LIN {X 0,Y 419.846,Z 525.532,A -85,B 0,C 180,E1 -10292.919,E2 -10292.919} C_VEL
LIN {X 0,Y 422.177,Z 533.001,A -85,B 0,C 180,E1 -10293.178,E2 -10293.178} C_VEL
LIN {X 0,Y 424.264,Z 542.34,A -85,B 0,C 180,E1 -10293.457,E2 -10293.457} C_VEL
LIN {X 0,Y 423.052,Z 632.06,A -85,B 0,C 180,E1 -10295.077,E2 -10295.077} C_VEL
LIN {X 0,Y 422.664,Z 645.822,A -85,B 0,C 180,E1 -10295.536,E2 -10295.536} C_VEL
LIN {X 0,Y 422.218,Z 658.144,A -85,B 0,C 180,E1 -10296.147,E2 -10296.147} C_VEL
LIN {X 0,Y 421.56,Z 670.212,A -85,B 0,C 180,E1 -10296.956,E2 -10296.956} C_VEL
LIN {X 0,Y 420.936,Z 680.638,A -85,B 0,C 180,E1 -10297.848,E2 -10297.848} C_VEL
LIN {X 0,Y 420.144,Z 691.488,A -85,B 0,C 180,E1 -10299.003,E2 -10299.003} C_VEL
LIN {X 0,Y 419.475,Z 700.404,A -85,B 0,C 180,E1 -10300.187,E2 -10300.187} C_VEL
LIN {X 0,Y 418.766,Z 709.277,A -85,B 0,C 180,E1 -10301.642,E2 -10301.642} C_VEL
LIN {X 0,Y 418.301,Z 715.982,A -85,B 0,C 180,E1 -10303.007,E2 -10303.007} C_VEL
LIN {X 0,Y 417.87,Z 721.394,A -85,B 0,C 180,E1 -10304.368,E2 -10304.368} C_VEL
LIN {X 0,Y 417.597,Z 725.629,A -85,B 0,C 180,E1 -10305.7,E2 -10305.7} C_VEL
LIN {X 0,Y 417.406,Z 728.908,A -85,B 0,C 180,E1 -10307.017,E2 -10307.017} C_VEL
LIN {X 0,Y 417.134,Z 732.231,A -85,B 0,C 180,E1 -10308.923,E2 -10308.923} C_VEL
LIN {X 0,Y 416.978,Z 733.892,A -85,B 0,C 180,E1 -10310.832,E2 -10310.832} C_VEL
LIN {X 0,Y 416.989,Z 734.062,A -85,B 0,C 180,E1 -10312.646,E2 -10312.646} C_VEL
LIN {X 0,Y 417.03,Z 733.266,A -85,B 0,C 180,E1 -10313.99,E2 -10313.99} C_VEL
LIN {X 0,Y 417.156,Z 731.24,A -85,B 0,C 180,E1 -10315.641,E2 -10315.641} C_VEL
LIN {X 0,Y 417.415,Z 727.732,A -85,B 0,C 180,E1 -10317.4,E2 -10317.4} C_VEL
LIN {X 0,Y 417.696,Z 722.842,A -85,B 0,C 180,E1 -10319.103,E2 -10319.103} C_VEL
LIN {X 0,Y 418.167,Z 716.254,A -85,B 0,C 180,E1 -10320.831,E2 -10320.831} C_VEL
LIN {X 0,Y 418.701,Z 708.425,A -85,B 0,C 180,E1 -10322.412,E2 -10322.412} C_VEL
LIN {X 0,Y 419.217,Z 701.022,A -85,B 0,C 180,E1 -10323.625,E2 -10323.625} C_VEL
LIN {X 0,Y 419.901,Z 691.588,A -85,B 0,C 180,E1 -10324.891,E2 -10324.891} C_VEL
LIN {X 0,Y 420.546,Z 681.763,A -85,B 0,C 180,E1 -10325.962,E2 -10325.962} C_VEL
LIN {X 0,Y 421.235,Z 670.138,A -85,B 0,C 180,E1 -10326.969,E2 -10326.969} C_VEL
LIN {X 0,Y 421.883,Z 657.865,A -85,B 0,C 180,E1 -10327.794,E2 -10327.794} C_VEL
LIN {X 0,Y 422.349,Z 645.01,A -85,B 0,C 180,E1 -10328.43,E2 -10328.43} C_VEL
LIN {X 0,Y 422.723,Z 631.3,A -85,B 0,C 180,E1 -10328.883,E2 -10328.883} C_VEL
LIN {X 0,Y 423.824,Z 551.136,A -85,B 0,C 180,E1 -10330.312,E2 -10330.312} C_VEL
LIN {X 0,Y 423.11,Z 547.36,A -85,B 0,C 180,E1 -10330.412,E2 -10330.412} C_VEL
LIN {X 0,Y 419.915,Z 541.784,A -85,B 0,C 180,E1 -10330.655,E2 -10330.655} C_VEL
LIN {X 0,Y 416.238,Z 536.306,A -85,B 0,C 180,E1 -10330.922,E2 -10330.922} C_VEL
LIN {X 0,Y 414.814,Z 532.618,A -85,B 0,C 180,E1 -10331.055,E2 -10331.055} C_VEL
LIN {X 0,Y 412.433,Z 524.509,A -85,B 0,C 180,E1 -10331.335,E2 -10331.335} C_VEL
LIN {X 0,Y 411.292,Z 518.255,A -85,B 0,C 180,E1 -10333.049,E2 -10333.049} C_VEL
LIN {X 0,Y 411.302,Z 518.255,A -85,B 0,C 180,E1 -10336.896,E2 -10336.896} C_VEL
LIN {X 0,Y 411.29,Z 518.249,A -85,B 0,C 180,E1 -10340.161,E2 -10340.161} C_VEL
LIN {X 0,Y 411.448,Z 518.233,A -85,B 0,C 180,E1 -10343.133,E2 -10343.133} C_VEL
LIN {X 0,Y 411.308,Z 518.251,A -85,B 0,C 180,E1 -10345.099,E2 -10345.099} C_VEL
LIN {X 0,Y 411.511,Z 518.221,A -85,B 0,C 180,E1 -10348.043,E2 -10348.043} C_VEL
LIN {X 0,Y 411.64,Z 518.205,A -85,B 0,C 180,E1 -10350,E2 -10350} C_VEL
LIN {X 0,Y 411.463,Z 518.235,A -85,B 0,C 180,E1 -10352.937,E2 -10352.937} C_VEL
LIN {X 0,Y 411.458,Z 518.234,A -85,B 0,C 180,E1 -10356.867,E2 -10356.867} C_VEL
LIN {X 0,Y 411.29,Z 518.249,A -85,B 0,C 180,E1 -10359.839,E2 -10359.839} C_VEL
LIN {X 0,Y 411.302,Z 518.253,A -85,B 0,C 180,E1 -10363.104,E2 -10363.104} C_VEL
LIN {X 0,Y 411.259,Z 518.259,A -85,B 0,C 180,E1 -10366.869,E2 -10366.869} C_VEL
LIN {X 0,Y 411.226,Z 518.256,A -85,B 0,C 180,E1 -10369.986,E2 -10369.986} C_VEL
LIN {X 0,Y 411.199,Z 518.266,A -85,B 0,C 180,E1 -10373.147,E2 -10373.147} C_VEL
LIN {X 0,Y 411.233,Z 518.257,A -85,B 0,C 180,E1 -10376.381,E2 -10376.381} C_VEL
LIN {X 0,Y 411.207,Z 518.26,A -85,B 0,C 180,E1 -10379.711,E2 -10379.711} C_VEL
LIN {X 0,Y 411.201,Z 518.266,A -85,B 0,C 180,E1 -10383.155,E2 -10383.155} C_VEL
LIN {X 0,Y 411.19,Z 518.263,A -85,B 0,C 180,E1 -10386.553,E2 -10386.553} C_VEL
LIN {X 0,Y 411.222,Z 518.258,A -85,B 0,C 180,E1 -10389.73,E2 -10389.73} C_VEL
LIN {X 0,Y 411.215,Z 518.265,A -85,B 0,C 180,E1 -10393.127,E2 -10393.127} C_VEL
LIN {X 0,Y 411.224,Z 518.257,A -85,B 0,C 180,E1 -10395.872,E2 -10395.872} C_VEL
LIN {X 0,Y 411.202,Z 518.263,A -85,B 0,C 180,E1 -10398.764,E2 -10398.764} C_VEL
LIN {X 0,Y 411.197,Z 518.26,A -85,B 0,C 180,E1 -10402.027,E2 -10402.027} C_VEL
LIN {X 0,Y 411.197,Z 518.262,A -85,B 0,C 180,E1 -10405.666,E2 -10405.666} C_VEL
LIN {X 0,Y 411.189,Z 518.268,A -85,B 0,C 180,E1 -10409.153,E2 -10409.153} C_VEL
LIN {X 0,Y 411.251,Z 518.255,A -85,B 0,C 180,E1 -10412.522,E2 -10412.522} C_VEL
LIN {X 0,Y 411.211,Z 518.259,A -85,B 0,C 180,E1 -10415.784,E2 -10415.784} C_VEL
LIN {X 0,Y 411.187,Z 518.267,A -85,B 0,C 180,E1 -10418.966,E2 -10418.966} C_VEL
LIN {X 0,Y 411.243,Z 518.254,A -85,B 0,C 180,E1 -10422.085,E2 -10422.085} C_VEL
LIN {X 0,Y 411.252,Z 518.261,A -85,B 0,C 180,E1 -10425.148,E2 -10425.148} C_VEL
LIN {X 0,Y 411.291,Z 518.248,A -85,B 0,C 180,E1 -10428.168,E2 -10428.168} C_VEL
LIN {X 0,Y 411.473,Z 518.226,A -85,B 0,C 180,E1 -10432.147,E2 -10432.147} C_VEL
LIN {X 0,Y 411.484,Z 518.224,A -85,B 0,C 180,E1 -10434.119,E2 -10434.119} C_VEL
LIN {X 0,Y 411.505,Z 518.222,A -85,B 0,C 180,E1 -10438.043,E2 -10438.043} C_VEL
LIN {X 0,Y 411.635,Z 518.206,A -85,B 0,C 180,E1 -10440,E2 -10440} C_VEL
LIN {X 0,Y 411.466,Z 518.231,A -85,B 0,C 180,E1 -10442.938,E2 -10442.938} C_VEL
LIN {X 0,Y 411.485,Z 518.225,A -85,B 0,C 180,E1 -10445.882,E2 -10445.882} C_VEL
LIN {X 0,Y 411.346,Z 518.245,A -85,B 0,C 180,E1 -10448.846,E2 -10448.846} C_VEL
LIN {X 0,Y 411.277,Z 518.251,A -85,B 0,C 180,E1 -10451.833,E2 -10451.833} C_VEL
LIN {X 0,Y 411.255,Z 518.256,A -85,B 0,C 180,E1 -10454.853,E2 -10454.853} C_VEL
LIN {X 0,Y 411.245,Z 518.255,A -85,B 0,C 180,E1 -10457.916,E2 -10457.916} C_VEL
LIN {X 0,Y 411.189,Z 518.266,A -85,B 0,C 180,E1 -10461.035,E2 -10461.035} C_VEL
LIN {X 0,Y 411.22,Z 518.257,A -85,B 0,C 180,E1 -10464.216,E2 -10464.216} C_VEL
LIN {X 0,Y 411.254,Z 518.258,A -85,B 0,C 180,E1 -10467.479,E2 -10467.479} C_VEL
LIN {X 0,Y 411.197,Z 518.263,A -85,B 0,C 180,E1 -10470.847,E2 -10470.847} C_VEL
LIN {X 0,Y 411.201,Z 518.26,A -85,B 0,C 180,E1 -10474.334,E2 -10474.334} C_VEL
LIN {X 0,Y 411.197,Z 518.261,A -85,B 0,C 180,E1 -10477.974,E2 -10477.974} C_VEL
LIN {X 0,Y 411.18,Z 518.262,A -85,B 0,C 180,E1 -10480.505,E2 -10480.505} C_VEL
LIN {X 0,Y 411.175,Z 518.268,A -85,B 0,C 180,E1 -10483.134,E2 -10483.134} C_VEL
LIN {X 0,Y 411.225,Z 518.258,A -85,B 0,C 180,E1 -10485.873,E2 -10485.873} C_VEL
LIN {X 0,Y 411.208,Z 518.26,A -85,B 0,C 180,E1 -10488.765,E2 -10488.765} C_VEL
LIN {X 0,Y 411.203,Z 518.26,A -85,B 0,C 180,E1 -10492.028,E2 -10492.028} C_VEL
LIN {X 0,Y 411.206,Z 518.265,A -85,B 0,C 180,E1 -10495.667,E2 -10495.667} C_VEL
LIN {X 0,Y 411.19,Z 518.266,A -85,B 0,C 180,E1 -10499.153,E2 -10499.153} C_VEL
LIN {X 0,Y 411.257,Z 518.466,A -85,B 0,C 180,E1 -10500.838,E2 -10500.838} C_VEL
LIN {X 0,Y 413.995,Z 531.161,A -85,B 0,C 180,E1 -10503.538,E2 -10503.538} C_VEL
LIN {X 0,Y 414.852,Z 536.822,A -85,B 0,C 180,E1 -10504.692,E2 -10504.692} C_VEL
LIN {X 0,Y 413.582,Z 554.54,A -85,B 0,C 180,E1 -10508.048,E2 -10508.048} C_VEL
LIN {X 0,Y 412.675,Z 568.68,A -85,B 0,C 180,E1 -10510.693,E2 -10510.693} C_VEL
LIN {X 0,Y 416.715,Z 597.46,A -85,B 0,C 180,E1 -10511.409,E2 -10511.409} C_VEL
LIN {X 0,Y 415.719,Z 677.331,A -85,B 0,C 180,E1 -10512.855,E2 -10512.855} C_VEL
LIN {X 0,Y 415.171,Z 690.524,A -85,B 0,C 180,E1 -10513.276,E2 -10513.276} C_VEL
LIN {X 0,Y 414.578,Z 702.127,A -85,B 0,C 180,E1 -10513.821,E2 -10513.821} C_VEL
LIN {X 0,Y 413.802,Z 714.608,A -85,B 0,C 180,E1 -10514.611,E2 -10514.611} C_VEL
LIN {X 0,Y 413.023,Z 726.338,A -85,B 0,C 180,E1 -10515.591,E2 -10515.591} C_VEL
LIN {X 0,Y 412.307,Z 737.064,A -85,B 0,C 180,E1 -10516.716,E2 -10516.716} C_VEL
LIN {X 0,Y 411.647,Z 746.405,A -85,B 0,C 180,E1 -10517.928,E2 -10517.928} C_VEL
LIN {X 0,Y 410.917,Z 755.563,A -85,B 0,C 180,E1 -10519.406,E2 -10519.406} C_VEL
LIN {X 0,Y 410.49,Z 762.952,A -85,B 0,C 180,E1 -10520.888,E2 -10520.888} C_VEL
LIN {X 0,Y 410.272,Z 767.956,A -85,B 0,C 180,E1 -10522.124,E2 -10522.124} C_VEL
LIN {X 0,Y 410.105,Z 773.082,A -85,B 0,C 180,E1 -10523.698,E2 -10523.698} C_VEL
LIN {X 0,Y 410.076,Z 776.523,A -85,B 0,C 180,E1 -10525.084,E2 -10525.084} C_VEL
LIN {X 0,Y 409.969,Z 778.431,A -85,B 0,C 180,E1 -10526.068,E2 -10526.068} C_VEL
LIN {X 0,Y 410.053,Z 779.888,A -85,B 0,C 180,E1 -10527.053,E2 -10527.053} C_VEL
LIN {X 0,Y 410.059,Z 780.907,A -85,B 0,C 180,E1 -10528.036,E2 -10528.036} C_VEL
LIN {X 0,Y 410.027,Z 781.527,A -85,B 0,C 180,E1 -10529.018,E2 -10529.018} C_VEL
LIN {X 0,Y 410.021,Z 781.753,A -85,B 0,C 180,E1 -10530,E2 -10530} C_VEL
LIN {X 0,Y 410.027,Z 781.545,A -85,B 0,C 180,E1 -10530.982,E2 -10530.982} C_VEL
LIN {X 0,Y 410.058,Z 780.924,A -85,B 0,C 180,E1 -10531.964,E2 -10531.964} C_VEL
LIN {X 0,Y 410.037,Z 779.904,A -85,B 0,C 180,E1 -10532.947,E2 -10532.947} C_VEL
LIN {X 0,Y 409.969,Z 778.476,A -85,B 0,C 180,E1 -10533.932,E2 -10533.932} C_VEL
LIN {X 0,Y 410.04,Z 775.484,A -85,B 0,C 180,E1 -10535.409,E2 -10535.409} C_VEL
LIN {X 0,Y 410.164,Z 771.443,A -85,B 0,C 180,E1 -10536.889,E2 -10536.889} C_VEL
LIN {X 0,Y 410.394,Z 765.241,A -85,B 0,C 180,E1 -10538.618,E2 -10538.618} C_VEL
LIN {X 0,Y 410.808,Z 758.468,A -85,B 0,C 180,E1 -10540.099,E2 -10540.099} C_VEL
LIN {X 0,Y 411.39,Z 750.078,A -85,B 0,C 180,E1 -10541.579,E2 -10541.579} C_VEL
LIN {X 0,Y 411.975,Z 741.495,A -85,B 0,C 180,E1 -10542.813,E2 -10542.813} C_VEL
LIN {X 0,Y 412.797,Z 731.164,A -85,B 0,C 180,E1 -10544.015,E2 -10544.015} C_VEL
LIN {X 0,Y 413.659,Z 719.054,A -85,B 0,C 180,E1 -10545.142,E2 -10545.142} C_VEL
LIN {X 0,Y 414.458,Z 707.157,A -85,B 0,C 180,E1 -10545.995,E2 -10545.995} C_VEL
LIN {X 0,Y 415.209,Z 694.838,A -85,B 0,C 180,E1 -10546.66,E2 -10546.66} C_VEL
LIN {X 0,Y 415.725,Z 683.207,A -85,B 0,C 180,E1 -10547.113,E2 -10547.113} C_VEL
LIN {X 0,Y 416.178,Z 669.616,A -85,B 0,C 180,E1 -10547.442,E2 -10547.442} C_VEL
LIN {X 0,Y 417.069,Z 597.113,A -85,B 0,C 180,E1 -10548.749,E2 -10548.749} C_VEL
LIN {X 0,Y 413.297,Z 571.021,A -85,B 0,C 180,E1 -10549.431,E2 -10549.431} C_VEL
LIN {X 0,Y 412.747,Z 567.355,A -85,B 0,C 180,E1 -10549.553,E2 -10549.553} C_VEL
LIN {X 0,Y 413.895,Z 550.559,A -85,B 0,C 180,E1 -10552.724,E2 -10552.724} C_VEL
LIN {X 0,Y 414.908,Z 537.081,A -85,B 0,C 180,E1 -10555.308,E2 -10555.308} C_VEL
LIN {X 0,Y 413.858,Z 530.206,A -85,B 0,C 180,E1 -10556.744,E2 -10556.744} C_VEL
LIN {X 0,Y 411.225,Z 518.262,A -85,B 0,C 180,E1 -10559.398,E2 -10559.398} C_VEL
LIN {X 0,Y 411.206,Z 518.267,A -85,B 0,C 180,E1 -10563.155,E2 -10563.155} C_VEL
LIN {X 0,Y 411.195,Z 518.27,A -85,B 0,C 180,E1 -10566.552,E2 -10566.552} C_VEL
LIN {X 0,Y 411.227,Z 518.259,A -85,B 0,C 180,E1 -10569.729,E2 -10569.729} C_VEL
LIN {X 0,Y 411.22,Z 518.262,A -85,B 0,C 180,E1 -10573.126,E2 -10573.126} C_VEL
LIN {X 0,Y 411.174,Z 518.264,A -85,B 0,C 180,E1 -10575.879,E2 -10575.879} C_VEL
LIN {X 0,Y 411.162,Z 518.271,A -85,B 0,C 180,E1 -10578.77,E2 -10578.77} C_VEL
LIN {X 0,Y 411.196,Z 518.262,A -85,B 0,C 180,E1 -10582.026,E2 -10582.026} C_VEL
LIN {X 0,Y 411.201,Z 518.258,A -85,B 0,C 180,E1 -10585.666,E2 -10585.666} C_VEL
LIN {X 0,Y 411.193,Z 518.263,A -85,B 0,C 180,E1 -10589.152,E2 -10589.152} C_VEL
LIN {X 0,Y 411.254,Z 518.255,A -85,B 0,C 180,E1 -10592.521,E2 -10592.521} C_VEL
LIN {X 0,Y 411.22,Z 518.254,A -85,B 0,C 180,E1 -10595.784,E2 -10595.784} C_VEL
LIN {X 0,Y 411.189,Z 518.263,A -85,B 0,C 180,E1 -10598.965,E2 -10598.965} C_VEL
LIN {X 0,Y 411.245,Z 518.255,A -85,B 0,C 180,E1 -10602.084,E2 -10602.084} C_VEL
LIN {X 0,Y 411.255,Z 518.257,A -85,B 0,C 180,E1 -10605.147,E2 -10605.147} C_VEL
LIN {X 0,Y 411.277,Z 518.252,A -85,B 0,C 180,E1 -10608.167,E2 -10608.167} C_VEL
LIN {X 0,Y 411.432,Z 518.233,A -85,B 0,C 180,E1 -10612.188,E2 -10612.188} C_VEL
LIN {X 0,Y 411.484,Z 518.222,A -85,B 0,C 180,E1 -10614.118,E2 -10614.118} C_VEL
LIN {X 0,Y 411.505,Z 518.222,A -85,B 0,C 180,E1 -10618.042,E2 -10618.042} C_VEL
LIN {X 0,Y 411.635,Z 518.205,A -85,B 0,C 180,E1 -10620,E2 -10620} C_VEL
LIN {X 0,Y 411.46,Z 518.232,A -85,B 0,C 180,E1 -10622.937,E2 -10622.937} C_VEL
LIN {X 0,Y 411.446,Z 518.23,A -85,B 0,C 180,E1 -10626.609,E2 -10626.609} C_VEL
LIN {X 0,Y 411.285,Z 518.252,A -85,B 0,C 180,E1 -10629.838,E2 -10629.838} C_VEL
LIN {X 0,Y 411.296,Z 518.254,A -85,B 0,C 180,E1 -10633.104,E2 -10633.104} C_VEL
LIN {X 0,Y 411.254,Z 518.26,A -85,B 0,C 180,E1 -10636.869,E2 -10636.869} C_VEL
LIN {X 0,Y 411.221,Z 518.26,A -85,B 0,C 180,E1 -10639.987,E2 -10639.987} C_VEL
LIN {X 0,Y 411.194,Z 518.27,A -85,B 0,C 180,E1 -10643.148,E2 -10643.148} C_VEL
LIN {X 0,Y 411.229,Z 518.266,A -85,B 0,C 180,E1 -10646.381,E2 -10646.381} C_VEL
LIN {X 0,Y 411.228,Z 518.262,A -85,B 0,C 180,E1 -10649.71,E2 -10649.71} C_VEL
LIN {X 0,Y 411.228,Z 518.326,A -85,B 0,C 180,E1 -10650.417,E2 -10650.417} C_VEL
LIN {X 0,Y 412.734,Z 525.88,A -85,B 0,C 180,E1 -10652.545,E2 -10652.545} C_VEL
LIN {X 0,Y 415.694,Z 534.839,A -85,B 0,C 180,E1 -10652.881,E2 -10652.881} C_VEL
LIN {X 0,Y 417.669,Z 543.921,A -85,B 0,C 180,E1 -10653.155,E2 -10653.155} C_VEL
LIN {X 0,Y 416.339,Z 631.969,A -85,B 0,C 180,E1 -10654.766,E2 -10654.766} C_VEL
LIN {X 0,Y 415.899,Z 645.587,A -85,B 0,C 180,E1 -10655.217,E2 -10655.217} C_VEL
LIN {X 0,Y 415.446,Z 658.415,A -85,B 0,C 180,E1 -10655.857,E2 -10655.857} C_VEL
LIN {X 0,Y 414.771,Z 670.154,A -85,B 0,C 180,E1 -10656.65,E2 -10656.65} C_VEL
LIN {X 0,Y 414.047,Z 681.808,A -85,B 0,C 180,E1 -10657.666,E2 -10657.666} C_VEL
LIN {X 0,Y 413.197,Z 692.747,A -85,B 0,C 180,E1 -10658.874,E2 -10658.874} C_VEL
LIN {X 0,Y 412.472,Z 701.767,A -85,B 0,C 180,E1 -10660.116,E2 -10660.116} C_VEL
LIN {X 0,Y 411.748,Z 710.41,A -85,B 0,C 180,E1 -10661.583,E2 -10661.583} C_VEL
LIN {X 0,Y 411.212,Z 717.61,A -85,B 0,C 180,E1 -10663.128,E2 -10663.128} C_VEL
LIN {X 0,Y 410.773,Z 722.895,A -85,B 0,C 180,E1 -10664.545,E2 -10664.545} C_VEL
LIN {X 0,Y 410.473,Z 727.125,A -85,B 0,C 180,E1 -10665.98,E2 -10665.98} C_VEL
LIN {X 0,Y 410.265,Z 730.393,A -85,B 0,C 180,E1 -10667.442,E2 -10667.442} C_VEL
LIN {X 0,Y 409.995,Z 733.205,A -85,B 0,C 180,E1 -10669.355,E2 -10669.355} C_VEL
LIN {X 0,Y 409.914,Z 734.224,A -85,B 0,C 180,E1 -10670.628,E2 -10670.628} C_VEL
LIN {X 0,Y 409.908,Z 734.58,A -85,B 0,C 180,E1 -10672.062,E2 -10672.062} C_VEL
LIN {X 0,Y 409.927,Z 733.943,A -85,B 0,C 180,E1 -10673.686,E2 -10673.686} C_VEL
LIN {X 0,Y 410.076,Z 731.835,A -85,B 0,C 180,E1 -10675.56,E2 -10675.56} C_VEL
LIN {X 0,Y 410.29,Z 729.042,A -85,B 0,C 180,E1 -10677.069,E2 -10677.069} C_VEL
LIN {X 0,Y 410.579,Z 724.387,A -85,B 0,C 180,E1 -10678.854,E2 -10678.854} C_VEL
LIN {X 0,Y 410.918,Z 719.504,A -85,B 0,C 180,E1 -10680.266,E2 -10680.266} C_VEL
LIN {X 0,Y 411.407,Z 713.295,A -85,B 0,C 180,E1 -10681.703,E2 -10681.703} C_VEL
LIN {X 0,Y 411.966,Z 705.678,A -85,B 0,C 180,E1 -10683.123,E2 -10683.123} C_VEL
LIN {X 0,Y 412.669,Z 696.527,A -85,B 0,C 180,E1 -10684.503,E2 -10684.503} C_VEL
LIN {X 0,Y 413.31,Z 687.21,A -85,B 0,C 180,E1 -10685.648,E2 -10685.648} C_VEL
LIN {X 0,Y 413.99,Z 676.911,A -85,B 0,C 180,E1 -10686.673,E2 -10686.673} C_VEL
LIN {X 0,Y 414.665,Z 665.353,A -85,B 0,C 180,E1 -10687.584,E2 -10687.584} C_VEL
LIN {X 0,Y 415.271,Z 653.102,A -85,B 0,C 180,E1 -10688.326,E2 -10688.326} C_VEL
LIN {X 0,Y 415.689,Z 640.417,A -85,B 0,C 180,E1 -10688.882,E2 -10688.882} C_VEL
LIN {X 0,Y 415.971,Z 627.154,A -85,B 0,C 180,E1 -10689.251,E2 -10689.251} C_VEL
LIN {X 0,Y 417.104,Z 543.216,A -85,B 0,C 180,E1 -10690.754,E2 -10690.754} C_VEL
LIN {X 0,Y 414.814,Z 532.618,A -85,B 0,C 180,E1 -10691.055,E2 -10691.055} C_VEL
LIN {X 0,Y 413.606,Z 529.676,A -85,B 0,C 180,E1 -10691.198,E2 -10691.198} C_VEL
LIN {X 0,Y 410.931,Z 526.466,A -85,B 0,C 180,E1 -10691.518,E2 -10691.518} C_VEL
LIN {X 0,Y 407.573,Z 523.715,A -85,B 0,C 180,E1 -10692.013,E2 -10692.013} C_VEL
LIN {X 0,Y 404.977,Z 521.31,A -85,B 0,C 180,E1 -10692.629,E2 -10692.629} C_VEL
LIN {X 0,Y 404.412,Z 520.066,A -85,B 0,C 180,E1 -10692.972,E2 -10692.972} C_VEL
LIN {X 0,Y 404.244,Z 519.133,A -85,B 0,C 180,E1 -10693.3,E2 -10693.3} C_VEL
LIN {X 0,Y 404.279,Z 519.129,A -85,B 0,C 180,E1 -10696.939,E2 -10696.939} C_VEL
LIN {X 0,Y 404.255,Z 519.125,A -85,B 0,C 180,E1 -10699.988,E2 -10699.988} C_VEL
LIN {X 0,Y 404.396,Z 519.113,A -85,B 0,C 180,E1 -10703.013,E2 -10703.013} C_VEL
LIN {X 0,Y 404.28,Z 519.128,A -85,B 0,C 180,E1 -10705.014,E2 -10705.014} C_VEL
LIN {X 0,Y 404.48,Z 519.097,A -85,B 0,C 180,E1 -10708.009,E2 -10708.009} C_VEL
LIN {X 0,Y 404.609,Z 519.081,A -85,B 0,C 180,E1 -10710,E2 -10710} C_VEL
LIN {X 0,Y 404.42,Z 519.111,A -85,B 0,C 180,E1 -10712.988,E2 -10712.988} C_VEL
LIN {X 0,Y 404.409,Z 519.113,A -85,B 0,C 180,E1 -10716.987,E2 -10716.987} C_VEL
LIN {X 0,Y 404.256,Z 519.125,A -85,B 0,C 180,E1 -10720.012,E2 -10720.012} C_VEL
LIN {X 0,Y 404.263,Z 519.128,A -85,B 0,C 180,E1 -10723.211,E2 -10723.211} C_VEL
LIN {X 0,Y 404.212,Z 519.138,A -85,B 0,C 180,E1 -10727.007,E2 -10727.007} C_VEL
LIN {X 0,Y 404.16,Z 519.138,A -85,B 0,C 180,E1 -10730.351,E2 -10730.351} C_VEL
LIN {X 0,Y 404.165,Z 519.138,A -85,B 0,C 180,E1 -10733.574,E2 -10733.574} C_VEL
LIN {X 0,Y 404.179,Z 519.135,A -85,B 0,C 180,E1 -10735.766,E2 -10735.766} C_VEL
LIN {X 0,Y 404.193,Z 519.133,A -85,B 0,C 180,E1 -10737.999,E2 -10737.999} C_VEL
LIN {X 0,Y 404.142,Z 519.141,A -85,B 0,C 180,E1 -10741.56,E2 -10741.56} C_VEL
LIN {X 0,Y 404.18,Z 519.142,A -85,B 0,C 180,E1 -10745.016,E2 -10745.016} C_VEL
LIN {X 0,Y 404.158,Z 519.141,A -85,B 0,C 180,E1 -10748.755,E2 -10748.755} C_VEL
LIN {X 0,Y 404.185,Z 519.135,A -85,B 0,C 180,E1 -10751.61,E2 -10751.61} C_VEL
LIN {X 0,Y 404.19,Z 519.135,A -85,B 0,C 180,E1 -10754.529,E2 -10754.529} C_VEL
LIN {X 0,Y 404.199,Z 519.136,A -85,B 0,C 180,E1 -10757.305,E2 -10757.305} C_VEL
LIN {X 0,Y 404.161,Z 519.137,A -85,B 0,C 180,E1 -10759.955,E2 -10759.955} C_VEL
LIN {X 0,Y 404.133,Z 519.147,A -85,B 0,C 180,E1 -10763.124,E2 -10763.124} C_VEL
LIN {X 0,Y 404.136,Z 519.14,A -85,B 0,C 180,E1 -10766.188,E2 -10766.188} C_VEL
LIN {X 0,Y 404.145,Z 519.14,A -85,B 0,C 180,E1 -10769.715,E2 -10769.715} C_VEL
LIN {X 0,Y 404.187,Z 519.141,A -85,B 0,C 180,E1 -10773.123,E2 -10773.123} C_VEL
LIN {X 0,Y 404.165,Z 519.141,A -85,B 0,C 180,E1 -10775.334,E2 -10775.334} C_VEL
LIN {X 0,Y 404.129,Z 519.142,A -85,B 0,C 180,E1 -10778.581,E2 -10778.581} C_VEL
LIN {X 0,Y 404.201,Z 519.133,A -85,B 0,C 180,E1 -10781.762,E2 -10781.762} C_VEL
LIN {X 0,Y 404.198,Z 519.136,A -85,B 0,C 180,E1 -10784.882,E2 -10784.882} C_VEL
LIN {X 0,Y 404.261,Z 519.124,A -85,B 0,C 180,E1 -10787.959,E2 -10787.959} C_VEL
LIN {X 0,Y 404.424,Z 519.104,A -85,B 0,C 180,E1 -10792.1,E2 -10792.1} C_VEL
LIN {X 0,Y 404.43,Z 519.103,A -85,B 0,C 180,E1 -10794.016,E2 -10794.016} C_VEL
LIN {X 0,Y 404.474,Z 519.098,A -85,B 0,C 180,E1 -10798.009,E2 -10798.009} C_VEL
LIN {X 0,Y 404.604,Z 519.082,A -85,B 0,C 180,E1 -10800,E2 -10800} C_VEL
LIN {X 0,Y 404.423,Z 519.109,A -85,B 0,C 180,E1 -10802.989,E2 -10802.989} C_VEL
LIN {X 0,Y 404.43,Z 519.104,A -85,B 0,C 180,E1 -10805.985,E2 -10805.985} C_VEL
LIN {X 0,Y 404.284,Z 519.126,A -85,B 0,C 180,E1 -10809.002,E2 -10809.002} C_VEL
LIN {X 0,Y 404.25,Z 519.126,A -85,B 0,C 180,E1 -10812.042,E2 -10812.042} C_VEL
LIN {X 0,Y 404.201,Z 519.138,A -85,B 0,C 180,E1 -10815.119,E2 -10815.119} C_VEL
LIN {X 0,Y 404.203,Z 519.131,A -85,B 0,C 180,E1 -10818.239,E2 -10818.239} C_VEL
LIN {X 0,Y 404.132,Z 519.146,A -85,B 0,C 180,E1 -10821.42,E2 -10821.42} C_VEL
LIN {X 0,Y 404.171,Z 519.137,A -85,B 0,C 180,E1 -10824.667,E2 -10824.667} C_VEL
LIN {X 0,Y 404.192,Z 519.133,A -85,B 0,C 180,E1 -10828,E2 -10828} C_VEL
LIN {X 0,Y 404.143,Z 519.143,A -85,B 0,C 180,E1 -10831.561,E2 -10831.561} C_VEL
LIN {X 0,Y 404.181,Z 519.138,A -85,B 0,C 180,E1 -10835.017,E2 -10835.017} C_VEL
LIN {X 0,Y 404.155,Z 519.139,A -85,B 0,C 180,E1 -10838.757,E2 -10838.757} C_VEL
LIN {X 0,Y 404.121,Z 519.146,A -85,B 0,C 180,E1 -10841.601,E2 -10841.601} C_VEL
LIN {X 0,Y 404.154,Z 519.138,A -85,B 0,C 180,E1 -10844.525,E2 -10844.525} C_VEL
LIN {X 0,Y 404.205,Z 519.138,A -85,B 0,C 180,E1 -10847.306,E2 -10847.306} C_VEL
LIN {X 0,Y 404.167,Z 519.137,A -85,B 0,C 180,E1 -10849.956,E2 -10849.956} C_VEL
LIN {X 0,Y 404.14,Z 519.144,A -85,B 0,C 180,E1 -10853.125,E2 -10853.125} C_VEL
LIN {X 0,Y 404.145,Z 519.142,A -85,B 0,C 180,E1 -10856.189,E2 -10856.189} C_VEL
LIN {X 0,Y 404.146,Z 519.144,A -85,B 0,C 180,E1 -10859.716,E2 -10859.716} C_VEL
LIN {X 0,Y 404.182,Z 519.154,A -85,B 0,C 180,E1 -10860.525,E2 -10860.525} C_VEL
LIN {X 0,Y 407.241,Z 533.536,A -85,B 0,C 180,E1 -10863.634,E2 -10863.634} C_VEL
LIN {X 0,Y 407.887,Z 539.01,A -85,B 0,C 180,E1 -10864.758,E2 -10864.758} C_VEL
LIN {X 0,Y 406.527,Z 556.798,A -85,B 0,C 180,E1 -10868.181,E2 -10868.181} C_VEL
LIN {X 0,Y 405.771,Z 568.442,A -85,B 0,C 180,E1 -10870.376,E2 -10870.376} C_VEL
LIN {X 0,Y 409.949,Z 597.889,A -85,B 0,C 180,E1 -10871.124,E2 -10871.124} C_VEL
LIN {X 0,Y 408.892,Z 677.36,A -85,B 0,C 180,E1 -10872.592,E2 -10872.592} C_VEL
LIN {X 0,Y 408.296,Z 691.166,A -85,B 0,C 180,E1 -10873.05,E2 -10873.05} C_VEL
LIN {X 0,Y 407.677,Z 702.501,A -85,B 0,C 180,E1 -10873.603,E2 -10873.603} C_VEL
LIN {X 0,Y 406.922,Z 713.946,A -85,B 0,C 180,E1 -10874.344,E2 -10874.344} C_VEL
LIN {X 0,Y 406.114,Z 725.731,A -85,B 0,C 180,E1 -10875.34,E2 -10875.34} C_VEL
LIN {X 0,Y 405.329,Z 737.011,A -85,B 0,C 180,E1 -10876.544,E2 -10876.544} C_VEL
LIN {X 0,Y 404.673,Z 745.875,A -85,B 0,C 180,E1 -10877.717,E2 -10877.717} C_VEL
LIN {X 0,Y 403.9,Z 755.059,A -85,B 0,C 180,E1 -10879.219,E2 -10879.219} C_VEL
LIN {X 0,Y 403.45,Z 762.468,A -85,B 0,C 180,E1 -10880.728,E2 -10880.728} C_VEL
LIN {X 0,Y 403.205,Z 767.487,A -85,B 0,C 180,E1 -10881.985,E2 -10881.985} C_VEL
LIN {X 0,Y 403,Z 773.074,A -85,B 0,C 180,E1 -10883.742,E2 -10883.742} C_VEL
LIN {X 0,Y 402.984,Z 776.082,A -85,B 0,C 180,E1 -10884.998,E2 -10884.998} C_VEL
LIN {X 0,Y 402.889,Z 777.997,A -85,B 0,C 180,E1 -10885.999,E2 -10885.999} C_VEL
LIN {X 0,Y 402.952,Z 779.463,A -85,B 0,C 180,E1 -10887.001,E2 -10887.001} C_VEL
LIN {X 0,Y 402.987,Z 780.489,A -85,B 0,C 180,E1 -10888.001,E2 -10888.001} C_VEL
LIN {X 0,Y 402.949,Z 781.112,A -85,B 0,C 180,E1 -10889.001,E2 -10889.001} C_VEL
LIN {X 0,Y 402.942,Z 781.342,A -85,B 0,C 180,E1 -10890,E2 -10890} C_VEL
LIN {X 0,Y 402.949,Z 781.142,A -85,B 0,C 180,E1 -10890.999,E2 -10890.999} C_VEL
LIN {X 0,Y 402.985,Z 780.524,A -85,B 0,C 180,E1 -10891.999,E2 -10891.999} C_VEL
LIN {X 0,Y 402.936,Z 779.503,A -85,B 0,C 180,E1 -10892.999,E2 -10892.999} C_VEL
LIN {X 0,Y 402.888,Z 778.079,A -85,B 0,C 180,E1 -10894.001,E2 -10894.001} C_VEL
LIN {X 0,Y 402.94,Z 775.09,A -85,B 0,C 180,E1 -10895.505,E2 -10895.505} C_VEL
LIN {X 0,Y 403.076,Z 771.053,A -85,B 0,C 180,E1 -10897.01,E2 -10897.01} C_VEL
LIN {X 0,Y 403.345,Z 764.863,A -85,B 0,C 180,E1 -10898.769,E2 -10898.769} C_VEL
LIN {X 0,Y 403.752,Z 758.104,A -85,B 0,C 180,E1 -10900.277,E2 -10900.277} C_VEL
LIN {X 0,Y 404.379,Z 749.734,A -85,B 0,C 180,E1 -10901.783,E2 -10901.783} C_VEL
LIN {X 0,Y 405.024,Z 741.18,A -85,B 0,C 180,E1 -10903.036,E2 -10903.036} C_VEL
LIN {X 0,Y 405.908,Z 730.638,A -85,B 0,C 180,E1 -10904.284,E2 -10904.284} C_VEL
LIN {X 0,Y 406.782,Z 718.793,A -85,B 0,C 180,E1 -10905.404,E2 -10905.404} C_VEL
LIN {X 0,Y 407.621,Z 706.962,A -85,B 0,C 180,E1 -10906.27,E2 -10906.27} C_VEL
LIN {X 0,Y 408.404,Z 694.717,A -85,B 0,C 180,E1 -10906.945,E2 -10906.945} C_VEL
LIN {X 0,Y 409.014,Z 682.313,A -85,B 0,C 180,E1 -10907.435,E2 -10907.435} C_VEL
LIN {X 0,Y 409.494,Z 668.321,A -85,B 0,C 180,E1 -10907.768,E2 -10907.768} C_VEL
LIN {X 0,Y 410.315,Z 597.245,A -85,B 0,C 180,E1 -10909.079,E2 -10909.079} C_VEL
LIN {X 0,Y 406.86,Z 573.145,A -85,B 0,C 180,E1 -10909.727,E2 -10909.727} C_VEL
LIN {X 0,Y 405.853,Z 566.857,A -85,B 0,C 180,E1 -10909.935,E2 -10909.935} C_VEL
LIN {X 0,Y 407.034,Z 550.286,A -85,B 0,C 180,E1 -10913.129,E2 -10913.129} C_VEL
LIN {X 0,Y 407.99,Z 538.122,A -85,B 0,C 180,E1 -10915.508,E2 -10915.508} C_VEL
LIN {X 0,Y 406.323,Z 528.631,A -85,B 0,C 180,E1 -10917.56,E2 -10917.56} C_VEL
LIN {X 0,Y 404.171,Z 519.142,A -85,B 0,C 180,E1 -10919.753,E2 -10919.753} C_VEL
LIN {X 0,Y 404.171,Z 519.144,A -85,B 0,C 180,E1 -10923.419,E2 -10923.419} C_VEL
LIN {X 0,Y 404.144,Z 519.146,A -85,B 0,C 180,E1 -10926.245,E2 -10926.245} C_VEL
LIN {X 0,Y 404.162,Z 519.142,A -85,B 0,C 180,E1 -10928.755,E2 -10928.755} C_VEL
LIN {X 0,Y 404.19,Z 519.136,A -85,B 0,C 180,E1 -10931.61,E2 -10931.61} C_VEL
LIN {X 0,Y 404.188,Z 519.14,A -85,B 0,C 180,E1 -10934.528,E2 -10934.528} C_VEL
LIN {X 0,Y 404.136,Z 519.14,A -85,B 0,C 180,E1 -10937.295,E2 -10937.295} C_VEL
LIN {X 0,Y 404.165,Z 519.137,A -85,B 0,C 180,E1 -10939.954,E2 -10939.954} C_VEL
LIN {X 0,Y 404.136,Z 519.142,A -85,B 0,C 180,E1 -10943.123,E2 -10943.123} C_VEL
LIN {X 0,Y 404.14,Z 519.139,A -85,B 0,C 180,E1 -10946.187,E2 -10946.187} C_VEL
LIN {X 0,Y 404.148,Z 519.139,A -85,B 0,C 180,E1 -10949.715,E2 -10949.715} C_VEL
LIN {X 0,Y 404.19,Z 519.138,A -85,B 0,C 180,E1 -10953.122,E2 -10953.122} C_VEL
LIN {X 0,Y 404.171,Z 519.134,A -85,B 0,C 180,E1 -10955.333,E2 -10955.333} C_VEL
LIN {X 0,Y 404.132,Z 519.145,A -85,B 0,C 180,E1 -10958.58,E2 -10958.58} C_VEL
LIN {X 0,Y 404.203,Z 519.132,A -85,B 0,C 180,E1 -10961.761,E2 -10961.761} C_VEL
LIN {X 0,Y 404.2,Z 519.139,A -85,B 0,C 180,E1 -10964.881,E2 -10964.881} C_VEL
LIN {X 0,Y 404.249,Z 519.127,A -85,B 0,C 180,E1 -10967.958,E2 -10967.958} C_VEL
LIN {X 0,Y 404.397,Z 519.109,A -85,B 0,C 180,E1 -10972.128,E2 -10972.128} C_VEL
LIN {X 0,Y 404.43,Z 519.101,A -85,B 0,C 180,E1 -10974.015,E2 -10974.015} C_VEL
LIN {X 0,Y 404.474,Z 519.098,A -85,B 0,C 180,E1 -10978.008,E2 -10978.008} C_VEL
LIN {X 0,Y 404.604,Z 519.081,A -85,B 0,C 180,E1 -10980,E2 -10980} C_VEL
LIN {X 0,Y 404.417,Z 519.109,A -85,B 0,C 180,E1 -10982.988,E2 -10982.988} C_VEL
LIN {X 0,Y 404.394,Z 519.108,A -85,B 0,C 180,E1 -10986.607,E2 -10986.607} C_VEL
LIN {X 0,Y 404.282,Z 519.126,A -85,B 0,C 180,E1 -10989.001,E2 -10989.001} C_VEL
LIN {X 0,Y 404.248,Z 519.128,A -85,B 0,C 180,E1 -10992.041,E2 -10992.041} C_VEL
LIN {X 0,Y 404.199,Z 519.139,A -85,B 0,C 180,E1 -10995.118,E2 -10995.118} C_VEL
LIN {X 0,Y 404.201,Z 519.135,A -85,B 0,C 180,E1 -10998.238,E2 -10998.238} C_VEL
LIN {X 0,Y 404.129,Z 519.148,A -85,B 0,C 180,E1 -11001.419,E2 -11001.419} C_VEL
LIN {X 0,Y 404.168,Z 519.144,A -85,B 0,C 180,E1 -11004.666,E2 -11004.666} C_VEL
LIN {X 0,Y 404.189,Z 519.141,A -85,B 0,C 180,E1 -11007.999,E2 -11007.999} C_VEL
LIN {X 0,Y 404.211,Z 519.237,A -85,B 0,C 180,E1 -11010.121,E2 -11010.121} C_VEL
LIN {X 0,Y 405.659,Z 526.375,A -85,B 0,C 180,E1 -11012.166,E2 -11012.166} C_VEL
LIN {X 0,Y 409.303,Z 537.008,A -85,B 0,C 180,E1 -11012.579,E2 -11012.579} C_VEL
LIN {X 0,Y 410.954,Z 544.278,A -85,B 0,C 180,E1 -11012.81,E2 -11012.81} C_VEL
LIN {X 0,Y 409.623,Z 632.401,A -85,B 0,C 180,E1 -11014.459,E2 -11014.459} C_VEL
LIN {X 0,Y 409.154,Z 646.089,A -85,B 0,C 180,E1 -11014.92,E2 -11014.92} C_VEL
LIN {X 0,Y 408.738,Z 658.091,A -85,B 0,C 180,E1 -11015.525,E2 -11015.525} C_VEL
LIN {X 0,Y 408.061,Z 669.579,A -85,B 0,C 180,E1 -11016.294,E2 -11016.294} C_VEL
LIN {X 0,Y 407.327,Z 680.603,A -85,B 0,C 180,E1 -11017.245,E2 -11017.245} C_VEL
LIN {X 0,Y 406.507,Z 690.936,A -85,B 0,C 180,E1 -11018.357,E2 -11018.357} C_VEL
LIN {X 0,Y 405.744,Z 700.274,A -85,B 0,C 180,E1 -11019.599,E2 -11019.599} C_VEL
LIN {X 0,Y 404.965,Z 708.795,A -85,B 0,C 180,E1 -11021.005,E2 -11021.005} C_VEL
LIN {X 0,Y 404.379,Z 715.708,A -85,B 0,C 180,E1 -11022.41,E2 -11022.41} C_VEL
LIN {X 0,Y 403.809,Z 722.404,A -85,B 0,C 180,E1 -11024.12,E2 -11024.12} C_VEL
LIN {X 0,Y 403.433,Z 727.471,A -85,B 0,C 180,E1 -11025.829,E2 -11025.829} C_VEL
LIN {X 0,Y 403.222,Z 730.498,A -85,B 0,C 180,E1 -11027.177,E2 -11027.177} C_VEL
LIN {X 0,Y 403.027,Z 732.765,A -85,B 0,C 180,E1 -11028.575,E2 -11028.575} C_VEL
LIN {X 0,Y 402.845,Z 734.36,A -85,B 0,C 180,E1 -11030.14,E2 -11030.14} C_VEL
LIN {X 0,Y 402.814,Z 734.972,A -85,B 0,C 180,E1 -11031.732,E2 -11031.732} C_VEL
LIN {X 0,Y 402.846,Z 734.414,A -85,B 0,C 180,E1 -11033.62,E2 -11033.62} C_VEL
LIN {X 0,Y 402.923,Z 733.005,A -85,B 0,C 180,E1 -11035.064,E2 -11035.064} C_VEL
LIN {X 0,Y 403.176,Z 730.189,A -85,B 0,C 180,E1 -11036.794,E2 -11036.794} C_VEL
LIN {X 0,Y 403.46,Z 725.812,A -85,B 0,C 180,E1 -11038.599,E2 -11038.599} C_VEL
LIN {X 0,Y 403.838,Z 720.911,A -85,B 0,C 180,E1 -11040.113,E2 -11040.113} C_VEL
LIN {X 0,Y 404.358,Z 714.255,A -85,B 0,C 180,E1 -11041.731,E2 -11041.731} C_VEL
LIN {X 0,Y 404.938,Z 706.784,A -85,B 0,C 180,E1 -11043.177,E2 -11043.177} C_VEL
LIN {X 0,Y 405.675,Z 697.548,A -85,B 0,C 180,E1 -11044.611,E2 -11044.611} C_VEL
LIN {X 0,Y 406.373,Z 687.891,A -85,B 0,C 180,E1 -11045.828,E2 -11045.828} C_VEL
LIN {X 0,Y 407.093,Z 677.614,A -85,B 0,C 180,E1 -11046.875,E2 -11046.875} C_VEL
LIN {X 0,Y 407.804,Z 665.97,A -85,B 0,C 180,E1 -11047.811,E2 -11047.811} C_VEL
LIN {X 0,Y 408.376,Z 654.37,A -85,B 0,C 180,E1 -11048.535,E2 -11048.535} C_VEL
LIN {X 0,Y 408.852,Z 641.984,A -85,B 0,C 180,E1 -11049.104,E2 -11049.104} C_VEL
LIN {X 0,Y 409.136,Z 629.518,A -85,B 0,C 180,E1 -11049.481,E2 -11049.481} C_VEL
LIN {X 0,Y 410.364,Z 544.174,A -85,B 0,C 180,E1 -11051.043,E2 -11051.043} C_VEL
LIN {X 0,Y 407.31,Z 531.119,A -85,B 0,C 180,E1 -11051.435,E2 -11051.435} C_VEL
LIN {X 0,Y 405.292,Z 524.809,A -85,B 0,C 180,E1 -11051.682,E2 -11051.682} C_VEL
LIN {X 0,Y 404.412,Z 520.066,A -85,B 0,C 180,E1 -11052.972,E2 -11052.972} C_VEL
LIN {X 0,Y 403.942,Z 519.243,A -85,B 0,C 180,E1 -11053.416,E2 -11053.416} C_VEL
LIN {X 0,Y 401.734,Z 519.445,A -85,B 0,C 180,E1 -11054.551,E2 -11054.551} C_VEL
LIN {X 0,Y 398.22,Z 520.018,A -85,B 0,C 180,E1 -11056.21,E2 -11056.21} C_VEL
LIN {X 0,Y 397.276,Z 520.01,A -85,B 0,C 180,E1 -11057.078,E2 -11057.078} C_VEL
LIN {X 0,Y 397.204,Z 520.003,A -85,B 0,C 180,E1 -11057.37,E2 -11057.37} C_VEL
LIN {X 0,Y 397.25,Z 520.004,A -85,B 0,C 180,E1 -11060.838,E2 -11060.838} C_VEL
LIN {X 0,Y 397.367,Z 519.983,A -85,B 0,C 180,E1 -11063.909,E2 -11063.909} C_VEL
LIN {X 0,Y 397.449,Z 519.973,A -85,B 0,C 180,E1 -11067.973,E2 -11067.973} C_VEL
LIN {X 0,Y 397.578,Z 519.957,A -85,B 0,C 180,E1 -11070,E2 -11070} C_VEL
LIN {X 0,Y 397.378,Z 519.988,A -85,B 0,C 180,E1 -11073.041,E2 -11073.041} C_VEL
LIN {X 0,Y 397.361,Z 519.989,A -85,B 0,C 180,E1 -11077.112,E2 -11077.112} C_VEL
LIN {X 0,Y 397.215,Z 520.002,A -85,B 0,C 180,E1 -11080.191,E2 -11080.191} C_VEL
LIN {X 0,Y 397.223,Z 520.004,A -85,B 0,C 180,E1 -11083.321,E2 -11083.321} C_VEL
LIN {X 0,Y 397.178,Z 520.012,A -85,B 0,C 180,E1 -11087.155,E2 -11087.155} C_VEL
LIN {X 0,Y 397.098,Z 520.021,A -85,B 0,C 180,E1 -11090.73,E2 -11090.73} C_VEL
LIN {X 0,Y 397.128,Z 520.013,A -85,B 0,C 180,E1 -11094.018,E2 -11094.018} C_VEL
LIN {X 0,Y 397.19,Z 520.008,A -85,B 0,C 180,E1 -11097.39,E2 -11097.39} C_VEL
LIN {X 0,Y 397.084,Z 520.024,A -85,B 0,C 180,E1 -11100.881,E2 -11100.881} C_VEL
LIN {X 0,Y 397.12,Z 520.015,A -85,B 0,C 180,E1 -11104.493,E2 -11104.493} C_VEL
LIN {X 0,Y 397.104,Z 520.016,A -85,B 0,C 180,E1 -11108.274,E2 -11108.274} C_VEL
LIN {X 0,Y 397.149,Z 520.01,A -85,B 0,C 180,E1 -11111.993,E2 -11111.993} C_VEL
LIN {X 0,Y 397.142,Z 520.019,A -85,B 0,C 180,E1 -11115.059,E2 -11115.059} C_VEL
LIN {X 0,Y 397.148,Z 520.01,A -85,B 0,C 180,E1 -11118.007,E2 -11118.007} C_VEL
LIN {X 0,Y 397.102,Z 520.017,A -85,B 0,C 180,E1 -11121.726,E2 -11121.726} C_VEL
LIN {X 0,Y 397.117,Z 520.017,A -85,B 0,C 180,E1 -11125.507,E2 -11125.507} C_VEL
LIN {X 0,Y 397.077,Z 520.027,A -85,B 0,C 180,E1 -11129.118,E2 -11129.118} C_VEL
LIN {X 0,Y 397.186,Z 520.007,A -85,B 0,C 180,E1 -11132.61,E2 -11132.61} C_VEL
LIN {X 0,Y 397.12,Z 520.014,A -85,B 0,C 180,E1 -11135.982,E2 -11135.982} C_VEL
LIN {X 0,Y 397.129,Z 520.014,A -85,B 0,C 180,E1 -11139.705,E2 -11139.705} C_VEL
LIN {X 0,Y 397.173,Z 520.011,A -85,B 0,C 180,E1 -11142.845,E2 -11142.845} C_VEL
LIN {X 0,Y 397.219,Z 520.004,A -85,B 0,C 180,E1 -11146.703,E2 -11146.703} C_VEL
LIN {X 0,Y 397.221,Z 520.002,A -85,B 0,C 180,E1 -11149.81,E2 -11149.81} C_VEL
LIN {X 0,Y 397.356,Z 519.988,A -85,B 0,C 180,E1 -11152.889,E2 -11152.889} C_VEL
LIN {X 0,Y 397.255,Z 520.001,A -85,B 0,C 180,E1 -11154.926,E2 -11154.926} C_VEL
LIN {X 0,Y 397.443,Z 519.974,A -85,B 0,C 180,E1 -11157.974,E2 -11157.974} C_VEL
LIN {X 0,Y 397.574,Z 519.958,A -85,B 0,C 180,E1 -11160.001,E2 -11160.001} C_VEL
LIN {X 0,Y 397.381,Z 519.986,A -85,B 0,C 180,E1 -11163.042,E2 -11163.042} C_VEL
LIN {X 0,Y 397.379,Z 519.982,A -85,B 0,C 180,E1 -11166.092,E2 -11166.092} C_VEL
LIN {X 0,Y 397.245,Z 520.005,A -85,B 0,C 180,E1 -11169.162,E2 -11169.162} C_VEL
LIN {X 0,Y 397.212,Z 520.002,A -85,B 0,C 180,E1 -11172.259,E2 -11172.259} C_VEL
LIN {X 0,Y 397.173,Z 520.013,A -85,B 0,C 180,E1 -11175.393,E2 -11175.393} C_VEL
LIN {X 0,Y 397.155,Z 520.01,A -85,B 0,C 180,E1 -11178.574,E2 -11178.574} C_VEL
LIN {X 0,Y 397.09,Z 520.019,A -85,B 0,C 180,E1 -11181.819,E2 -11181.819} C_VEL
LIN {X 0,Y 397.15,Z 520.015,A -85,B 0,C 180,E1 -11185.133,E2 -11185.133} C_VEL
LIN {X 0,Y 397.158,Z 520.011,A -85,B 0,C 180,E1 -11187.777,E2 -11187.777} C_VEL
LIN {X 0,Y 397.083,Z 520.021,A -85,B 0,C 180,E1 -11190.883,E2 -11190.883} C_VEL
LIN {X 0,Y 397.121,Z 520.014,A -85,B 0,C 180,E1 -11194.494,E2 -11194.494} C_VEL
LIN {X 0,Y 397.103,Z 520.016,A -85,B 0,C 180,E1 -11198.276,E2 -11198.276} C_VEL
LIN {X 0,Y 397.087,Z 520.02,A -85,B 0,C 180,E1 -11200.91,E2 -11200.91} C_VEL
LIN {X 0,Y 397.102,Z 520.02,A -85,B 0,C 180,E1 -11203.649,E2 -11203.649} C_VEL
LIN {X 0,Y 397.158,Z 520.009,A -85,B 0,C 180,E1 -11206.513,E2 -11206.513} C_VEL
LIN {X 0,Y 397.122,Z 520.019,A -85,B 0,C 180,E1 -11209.552,E2 -11209.552} C_VEL
LIN {X 0,Y 397.098,Z 520.018,A -85,B 0,C 180,E1 -11212.791,E2 -11212.791} C_VEL
LIN {X 0,Y 397.118,Z 520.018,A -85,B 0,C 180,E1 -11216.283,E2 -11216.283} C_VEL
LIN {X 0,Y 397.122,Z 520.018,A -85,B 0,C 180,E1 -11220.23,E2 -11220.23} C_VEL
LIN {X 0,Y 400.113,Z 533.895,A -85,B 0,C 180,E1 -11223.304,E2 -11223.304} C_VEL
LIN {X 0,Y 400.97,Z 539.897,A -85,B 0,C 180,E1 -11224.57,E2 -11224.57} C_VEL
LIN {X 0,Y 399.559,Z 557.675,A -85,B 0,C 180,E1 -11228.052,E2 -11228.052} C_VEL
LIN {X 0,Y 398.839,Z 567.91,A -85,B 0,C 180,E1 -11230.038,E2 -11230.038} C_VEL
LIN {X 0,Y 403.153,Z 598.829,A -85,B 0,C 180,E1 -11230.844,E2 -11230.844} C_VEL
LIN {X 0,Y 402.061,Z 677.13,A -85,B 0,C 180,E1 -11232.32,E2 -11232.32} C_VEL
LIN {X 0,Y 401.46,Z 690.881,A -85,B 0,C 180,E1 -11232.785,E2 -11232.785} C_VEL
LIN {X 0,Y 400.783,Z 702.755,A -85,B 0,C 180,E1 -11233.379,E2 -11233.379} C_VEL
LIN {X 0,Y 399.922,Z 714.822,A -85,B 0,C 180,E1 -11234.194,E2 -11234.194} C_VEL
LIN {X 0,Y 399.103,Z 726.371,A -85,B 0,C 180,E1 -11235.207,E2 -11235.207} C_VEL
LIN {X 0,Y 398.348,Z 736.837,A -85,B 0,C 180,E1 -11236.356,E2 -11236.356} C_VEL
LIN {X 0,Y 397.687,Z 745.316,A -85,B 0,C 180,E1 -11237.498,E2 -11237.498} C_VEL
LIN {X 0,Y 396.866,Z 754.537,A -85,B 0,C 180,E1 -11239.026,E2 -11239.026} C_VEL
LIN {X 0,Y 396.413,Z 761.974,A -85,B 0,C 180,E1 -11240.561,E2 -11240.561} C_VEL
LIN {X 0,Y 396.058,Z 768.787,A -85,B 0,C 180,E1 -11242.352,E2 -11242.352} C_VEL
LIN {X 0,Y 395.911,Z 773.275,A -85,B 0,C 180,E1 -11243.886,E2 -11243.886} C_VEL
LIN {X 0,Y 395.893,Z 775.64,A -85,B 0,C 180,E1 -11244.908,E2 -11244.908} C_VEL
LIN {X 0,Y 395.812,Z 777.562,A -85,B 0,C 180,E1 -11245.927,E2 -11245.927} C_VEL
LIN {X 0,Y 395.852,Z 779.038,A -85,B 0,C 180,E1 -11246.947,E2 -11246.947} C_VEL
LIN {X 0,Y 395.916,Z 780.07,A -85,B 0,C 180,E1 -11247.965,E2 -11247.965} C_VEL
LIN {X 0,Y 395.875,Z 780.697,A -85,B 0,C 180,E1 -11248.983,E2 -11248.983} C_VEL
LIN {X 0,Y 395.864,Z 780.93,A -85,B 0,C 180,E1 -11250,E2 -11250} C_VEL
LIN {X 0,Y 395.874,Z 780.739,A -85,B 0,C 180,E1 -11251.017,E2 -11251.017} C_VEL
LIN {X 0,Y 395.913,Z 780.124,A -85,B 0,C 180,E1 -11252.035,E2 -11252.035} C_VEL
LIN {X 0,Y 395.837,Z 779.106,A -85,B 0,C 180,E1 -11253.053,E2 -11253.053} C_VEL
LIN {X 0,Y 395.809,Z 777.687,A -85,B 0,C 180,E1 -11254.073,E2 -11254.073} C_VEL
LIN {X 0,Y 395.838,Z 774.212,A -85,B 0,C 180,E1 -11255.819,E2 -11255.819} C_VEL
LIN {X 0,Y 396.057,Z 769.074,A -85,B 0,C 180,E1 -11257.648,E2 -11257.648} C_VEL
LIN {X 0,Y 396.414,Z 762.442,A -85,B 0,C 180,E1 -11259.438,E2 -11259.438} C_VEL
LIN {X 0,Y 396.896,Z 755.179,A -85,B 0,C 180,E1 -11260.973,E2 -11260.973} C_VEL
LIN {X 0,Y 397.712,Z 746.165,A -85,B 0,C 180,E1 -11262.502,E2 -11262.502} C_VEL
LIN {X 0,Y 398.489,Z 736.719,A -85,B 0,C 180,E1 -11263.802,E2 -11263.802} C_VEL
LIN {X 0,Y 399.291,Z 726.733,A -85,B 0,C 180,E1 -11264.917,E2 -11264.917} C_VEL
LIN {X 0,Y 400.155,Z 715.431,A -85,B 0,C 180,E1 -11265.927,E2 -11265.927} C_VEL
LIN {X 0,Y 401.074,Z 702.781,A -85,B 0,C 180,E1 -11266.805,E2 -11266.805} C_VEL
LIN {X 0,Y 401.815,Z 689.776,A -85,B 0,C 180,E1 -11267.462,E2 -11267.462} C_VEL
LIN {X 0,Y 402.543,Z 675.997,A -85,B 0,C 180,E1 -11267.921,E2 -11267.921} C_VEL
LIN {X 0,Y 403.649,Z 598.109,A -85,B 0,C 180,E1 -11269.407,E2 -11269.407} C_VEL
LIN {X 0,Y 400.392,Z 575.093,A -85,B 0,C 180,E1 -11270.04,E2 -11270.04} C_VEL
LIN {X 0,Y 398.989,Z 566.581,A -85,B 0,C 180,E1 -11270.29,E2 -11270.29} C_VEL
LIN {X 0,Y 400.21,Z 550.017,A -85,B 0,C 180,E1 -11273.547,E2 -11273.547} C_VEL
LIN {X 0,Y 401.07,Z 539.239,A -85,B 0,C 180,E1 -11275.702,E2 -11275.702} C_VEL
LIN {X 0,Y 399.103,Z 528.633,A -85,B 0,C 180,E1 -11278.056,E2 -11278.056} C_VEL
LIN {X 0,Y 397.114,Z 520.021,A -85,B 0,C 180,E1 -11280.118,E2 -11280.118} C_VEL
LIN {X 0,Y 397.118,Z 520.023,A -85,B 0,C 180,E1 -11283.717,E2 -11283.717} C_VEL
LIN {X 0,Y 397.098,Z 520.021,A -85,B 0,C 180,E1 -11287.209,E2 -11287.209} C_VEL
LIN {X 0,Y 397.122,Z 520.019,A -85,B 0,C 180,E1 -11290.448,E2 -11290.448} C_VEL
LIN {X 0,Y 397.158,Z 520.012,A -85,B 0,C 180,E1 -11293.639,E2 -11293.639} C_VEL
LIN {X 0,Y 397.103,Z 520.022,A -85,B 0,C 180,E1 -11296.519,E2 -11296.519} C_VEL
LIN {X 0,Y 397.111,Z 520.017,A -85,B 0,C 180,E1 -11300.422,E2 -11300.422} C_VEL
LIN {X 0,Y 397.105,Z 520.018,A -85,B 0,C 180,E1 -11304.264,E2 -11304.264} C_VEL
LIN {X 0,Y 397.11,Z 520.018,A -85,B 0,C 180,E1 -11306.726,E2 -11306.726} C_VEL
LIN {X 0,Y 397.128,Z 520.015,A -85,B 0,C 180,E1 -11310.296,E2 -11310.296} C_VEL
LIN {X 0,Y 397.189,Z 520.006,A -85,B 0,C 180,E1 -11312.609,E2 -11312.609} C_VEL
LIN {X 0,Y 397.126,Z 520.01,A -85,B 0,C 180,E1 -11315.981,E2 -11315.981} C_VEL
LIN {X 0,Y 397.132,Z 520.011,A -85,B 0,C 180,E1 -11319.704,E2 -11319.704} C_VEL
LIN {X 0,Y 397.175,Z 520.008,A -85,B 0,C 180,E1 -11322.844,E2 -11322.844} C_VEL
LIN {X 0,Y 397.219,Z 520.002,A -85,B 0,C 180,E1 -11326.678,E2 -11326.678} C_VEL
LIN {X 0,Y 397.211,Z 520,A -85,B 0,C 180,E1 -11329.808,E2 -11329.808} C_VEL
LIN {X 0,Y 397.346,Z 519.989,A -85,B 0,C 180,E1 -11332.887,E2 -11332.887} C_VEL
LIN {X 0,Y 397.254,Z 520.001,A -85,B 0,C 180,E1 -11334.925,E2 -11334.925} C_VEL
LIN {X 0,Y 397.443,Z 519.974,A -85,B 0,C 180,E1 -11337.973,E2 -11337.973} C_VEL
LIN {X 0,Y 397.574,Z 519.957,A -85,B 0,C 180,E1 -11339.999,E2 -11339.999} C_VEL
LIN {X 0,Y 397.375,Z 519.985,A -85,B 0,C 180,E1 -11343.041,E2 -11343.041} C_VEL
LIN {X 0,Y 397.346,Z 519.986,A -85,B 0,C 180,E1 -11346.602,E2 -11346.602} C_VEL
LIN {X 0,Y 397.244,Z 520.002,A -85,B 0,C 180,E1 -11349.162,E2 -11349.162} C_VEL
LIN {X 0,Y 397.211,Z 520.005,A -85,B 0,C 180,E1 -11352.258,E2 -11352.258} C_VEL
LIN {X 0,Y 397.171,Z 520.012,A -85,B 0,C 180,E1 -11355.392,E2 -11355.392} C_VEL
LIN {X 0,Y 397.153,Z 520.014,A -85,B 0,C 180,E1 -11358.573,E2 -11358.573} C_VEL
LIN {X 0,Y 397.087,Z 520.023,A -85,B 0,C 180,E1 -11361.818,E2 -11361.818} C_VEL
LIN {X 0,Y 397.148,Z 520.018,A -85,B 0,C 180,E1 -11365.132,E2 -11365.132} C_VEL
LIN {X 0,Y 397.155,Z 520.019,A -85,B 0,C 180,E1 -11367.777,E2 -11367.777} C_VEL
LIN {X 0,Y 397.152,Z 520.057,A -85,B 0,C 180,E1 -11369.78,E2 -11369.78} C_VEL
LIN {X 0,Y 398.544,Z 526.764,A -85,B 0,C 180,E1 -11371.753,E2 -11371.753} C_VEL
LIN {X 0,Y 402.817,Z 538.833,A -85,B 0,C 180,E1 -11372.253,E2 -11372.253} C_VEL
LIN {X 0,Y 404.397,Z 546.799,A -85,B 0,C 180,E1 -11372.5,E2 -11372.5} C_VEL
LIN {X 0,Y 402.904,Z 633.211,A -85,B 0,C 180,E1 -11374.146,E2 -11374.146} C_VEL
LIN {X 0,Y 402.445,Z 646.829,A -85,B 0,C 180,E1 -11374.62,E2 -11374.62} C_VEL
LIN {X 0,Y 401.982,Z 658.77,A -85,B 0,C 180,E1 -11375.236,E2 -11375.236} C_VEL
LIN {X 0,Y 401.251,Z 670.55,A -85,B 0,C 180,E1 -11376.048,E2 -11376.048} C_VEL
LIN {X 0,Y 400.424,Z 682.393,A -85,B 0,C 180,E1 -11377.108,E2 -11377.108} C_VEL
LIN {X 0,Y 399.627,Z 691.751,A -85,B 0,C 180,E1 -11378.149,E2 -11378.149} C_VEL
LIN {X 0,Y 398.829,Z 700.758,A -85,B 0,C 180,E1 -11379.373,E2 -11379.373} C_VEL
LIN {X 0,Y 398.023,Z 709.208,A -85,B 0,C 180,E1 -11380.792,E2 -11380.792} C_VEL
LIN {X 0,Y 397.381,Z 716.144,A -85,B 0,C 180,E1 -11382.225,E2 -11382.225} C_VEL
LIN {X 0,Y 396.895,Z 721.822,A -85,B 0,C 180,E1 -11383.676,E2 -11383.676} C_VEL
LIN {X 0,Y 396.56,Z 726.407,A -85,B 0,C 180,E1 -11385.144,E2 -11385.144} C_VEL
LIN {X 0,Y 396.252,Z 730.051,A -85,B 0,C 180,E1 -11386.65,E2 -11386.65} C_VEL
LIN {X 0,Y 396.002,Z 732.76,A -85,B 0,C 180,E1 -11388.192,E2 -11388.192} C_VEL
LIN {X 0,Y 395.753,Z 734.906,A -85,B 0,C 180,E1 -11390.261,E2 -11390.261} C_VEL
LIN {X 0,Y 395.744,Z 735.365,A -85,B 0,C 180,E1 -11391.571,E2 -11391.571} C_VEL
LIN {X 0,Y 395.724,Z 735.125,A -85,B 0,C 180,E1 -11393.052,E2 -11393.052} C_VEL
LIN {X 0,Y 395.829,Z 733.791,A -85,B 0,C 180,E1 -11394.758,E2 -11394.758} C_VEL
LIN {X 0,Y 396.055,Z 731.021,A -85,B 0,C 180,E1 -11396.627,E2 -11396.627} C_VEL
LIN {X 0,Y 396.345,Z 727.208,A -85,B 0,C 180,E1 -11398.334,E2 -11398.334} C_VEL
LIN {X 0,Y 396.654,Z 723.243,A -85,B 0,C 180,E1 -11399.672,E2 -11399.672} C_VEL
LIN {X 0,Y 397.096,Z 717.737,A -85,B 0,C 180,E1 -11401.166,E2 -11401.166} C_VEL
LIN {X 0,Y 397.603,Z 710.99,A -85,B 0,C 180,E1 -11402.641,E2 -11402.641} C_VEL
LIN {X 0,Y 398.32,Z 702.439,A -85,B 0,C 180,E1 -11404.137,E2 -11404.137} C_VEL
LIN {X 0,Y 399.155,Z 692.336,A -85,B 0,C 180,E1 -11405.559,E2 -11405.559} C_VEL
LIN {X 0,Y 399.884,Z 682.146,A -85,B 0,C 180,E1 -11406.707,E2 -11406.707} C_VEL
LIN {X 0,Y 400.621,Z 671.371,A -85,B 0,C 180,E1 -11407.679,E2 -11407.679} C_VEL
LIN {X 0,Y 401.339,Z 658.902,A -85,B 0,C 180,E1 -11408.559,E2 -11408.559} C_VEL
LIN {X 0,Y 401.903,Z 645.904,A -85,B 0,C 180,E1 -11409.228,E2 -11409.228} C_VEL
LIN {X 0,Y 402.287,Z 632.319,A -85,B 0,C 180,E1 -11409.698,E2 -11409.698} C_VEL
LIN {X 0,Y 403.608,Z 545.176,A -85,B 0,C 180,E1 -11411.338,E2 -11411.338} C_VEL
LIN {X 0,Y 400.885,Z 533.475,A -85,B 0,C 180,E1 -11411.697,E2 -11411.697} C_VEL
LIN {X 0,Y 398.168,Z 525.195,A -85,B 0,C 180,E1 -11412.021,E2 -11412.021} C_VEL
LIN {X 0,Y 397.19,Z 520.01,A -85,B 0,C 180,E1 -11413.47,E2 -11413.47} C_VEL
LIN {X 0,Y 397.225,Z 520.006,A -85,B 0,C 180,E1 -11416.703,E2 -11416.703} C_VEL
LIN {X 0,Y 397.204,Z 520.003,A -85,B 0,C 180,E1 -11417.37,E2 -11417.37} C_VEL
LIN {X 0,Y 396.548,Z 520.087,A -85,B 0,C 180,E1 -11418.216,E2 -11418.216} C_VEL
LIN {X 0,Y 393.703,Z 520.44,A -85,B 0,C 180,E1 -11419.592,E2 -11419.592} C_VEL
LIN {X 0,Y 391.321,Z 520.741,A -85,B 0,C 180,E1 -11420.703,E2 -11420.703} C_VEL
LIN {X 0,Y 390.342,Z 520.859,A -85,B 0,C 180,E1 -11421.562,E2 -11421.562} C_VEL
LIN {X 0,Y 390.285,Z 520.865,A -85,B 0,C 180,E1 -11421.853,E2 -11421.853} C_VEL
LIN {X 0,Y 390.223,Z 520.879,A -85,B 0,C 180,E1 -11424.834,E2 -11424.834} C_VEL
LIN {X 0,Y 390.418,Z 520.849,A -85,B 0,C 180,E1 -11427.937,E2 -11427.937} C_VEL
LIN {X 0,Y 390.547,Z 520.833,A -85,B 0,C 180,E1 -11430,E2 -11430} C_VEL
LIN {X 0,Y 390.312,Z 520.867,A -85,B 0,C 180,E1 -11433.096,E2 -11433.096} C_VEL
LIN {X 0,Y 390.328,Z 520.86,A -85,B 0,C 180,E1 -11436.202,E2 -11436.202} C_VEL
LIN {X 0,Y 390.311,Z 520.863,A -85,B 0,C 180,E1 -11438.282,E2 -11438.282} C_VEL
LIN {X 0,Y 390.168,Z 520.882,A -85,B 0,C 180,E1 -11442.483,E2 -11442.483} C_VEL
LIN {X 0,Y 390.136,Z 520.884,A -85,B 0,C 180,E1 -11445.677,E2 -11445.677} C_VEL
LIN {X 0,Y 390.102,Z 520.895,A -85,B 0,C 180,E1 -11448.922,E2 -11448.922} C_VEL
LIN {X 0,Y 390.036,Z 520.897,A -85,B 0,C 180,E1 -11452.234,E2 -11452.234} C_VEL
LIN {X 0,Y 390.114,Z 520.887,A -85,B 0,C 180,E1 -11455.743,E2 -11455.743} C_VEL
LIN {X 0,Y 390.062,Z 520.899,A -85,B 0,C 180,E1 -11459.108,E2 -11459.108} C_VEL
LIN {X 0,Y 390.05,Z 520.898,A -85,B 0,C 180,E1 -11462.72,E2 -11462.72} C_VEL
LIN {X 0,Y 390.052,Z 520.895,A -85,B 0,C 180,E1 -11465.825,E2 -11465.825} C_VEL
LIN {X 0,Y 390.069,Z 520.897,A -85,B 0,C 180,E1 -11469.219,E2 -11469.219} C_VEL
LIN {X 0,Y 390.114,Z 520.887,A -85,B 0,C 180,E1 -11472.386,E2 -11472.386} C_VEL
LIN {X 0,Y 390.109,Z 520.891,A -85,B 0,C 180,E1 -11475.365,E2 -11475.365} C_VEL
LIN {X 0,Y 390.097,Z 520.889,A -85,B 0,C 180,E1 -11478.196,E2 -11478.196} C_VEL
LIN {X 0,Y 390.088,Z 520.895,A -85,B 0,C 180,E1 -11480.908,E2 -11480.908} C_VEL
LIN {X 0,Y 390.077,Z 520.895,A -85,B 0,C 180,E1 -11484.793,E2 -11484.793} C_VEL
LIN {X 0,Y 390.019,Z 520.9,A -85,B 0,C 180,E1 -11488.496,E2 -11488.496} C_VEL
LIN {X 0,Y 390.109,Z 520.887,A -85,B 0,C 180,E1 -11492.07,E2 -11492.07} C_VEL
LIN {X 0,Y 390.068,Z 520.895,A -85,B 0,C 180,E1 -11495.519,E2 -11495.519} C_VEL
LIN {X 0,Y 390.046,Z 520.899,A -85,B 0,C 180,E1 -11498.878,E2 -11498.878} C_VEL
LIN {X 0,Y 390.119,Z 520.886,A -85,B 0,C 180,E1 -11502.167,E2 -11502.167} C_VEL
LIN {X 0,Y 390.137,Z 520.888,A -85,B 0,C 180,E1 -11505.393,E2 -11505.393} C_VEL
LIN {X 0,Y 390.15,Z 520.883,A -85,B 0,C 180,E1 -11508.572,E2 -11508.572} C_VEL
LIN {X 0,Y 390.335,Z 520.859,A -85,B 0,C 180,E1 -11511.993,E2 -11511.993} C_VEL
LIN {X 0,Y 390.226,Z 520.876,A -85,B 0,C 180,E1 -11514.834,E2 -11514.834} C_VEL
LIN {X 0,Y 390.412,Z 520.85,A -85,B 0,C 180,E1 -11517.937,E2 -11517.937} C_VEL
LIN {X 0,Y 390.543,Z 520.833,A -85,B 0,C 180,E1 -11520.001,E2 -11520.001} C_VEL
LIN {X 0,Y 390.341,Z 520.864,A -85,B 0,C 180,E1 -11523.097,E2 -11523.097} C_VEL
LIN {X 0,Y 390.33,Z 520.86,A -85,B 0,C 180,E1 -11526.202,E2 -11526.202} C_VEL
LIN {X 0,Y 390.198,Z 520.882,A -85,B 0,C 180,E1 -11529.329,E2 -11529.329} C_VEL
LIN {X 0,Y 390.164,Z 520.881,A -85,B 0,C 180,E1 -11532.484,E2 -11532.484} C_VEL
LIN {X 0,Y 390.133,Z 520.887,A -85,B 0,C 180,E1 -11535.678,E2 -11535.678} C_VEL
LIN {X 0,Y 390.098,Z 520.892,A -85,B 0,C 180,E1 -11538.923,E2 -11538.923} C_VEL
LIN {X 0,Y 390.033,Z 520.897,A -85,B 0,C 180,E1 -11542.235,E2 -11542.235} C_VEL
LIN {X 0,Y 390.113,Z 520.889,A -85,B 0,C 180,E1 -11545.744,E2 -11545.744} C_VEL
LIN {X 0,Y 390.061,Z 520.898,A -85,B 0,C 180,E1 -11549.11,E2 -11549.11} C_VEL
LIN {X 0,Y 390.051,Z 520.896,A -85,B 0,C 180,E1 -11552.721,E2 -11552.721} C_VEL
LIN {X 0,Y 390.053,Z 520.896,A -85,B 0,C 180,E1 -11555.827,E2 -11555.827} C_VEL
LIN {X 0,Y 390.069,Z 520.898,A -85,B 0,C 180,E1 -11559.22,E2 -11559.22} C_VEL
LIN {X 0,Y 390.041,Z 520.896,A -85,B 0,C 180,E1 -11562.375,E2 -11562.375} C_VEL
LIN {X 0,Y 390.1,Z 520.889,A -85,B 0,C 180,E1 -11566.108,E2 -11566.108} C_VEL
LIN {X 0,Y 390.081,Z 520.896,A -85,B 0,C 180,E1 -11569.175,E2 -11569.175} C_VEL
LIN {X 0,Y 390.046,Z 520.895,A -85,B 0,C 180,E1 -11572.449,E2 -11572.449} C_VEL
LIN {X 0,Y 390.068,Z 520.897,A -85,B 0,C 180,E1 -11576.046,E2 -11576.046} C_VEL
LIN {X 0,Y 390.059,Z 520.978,A -85,B 0,C 180,E1 -11579.966,E2 -11579.966} C_VEL
LIN {X 0,Y 393.146,Z 535.187,A -85,B 0,C 180,E1 -11583.169,E2 -11583.169} C_VEL
LIN {X 0,Y 394.027,Z 540.761,A -85,B 0,C 180,E1 -11584.372,E2 -11584.372} C_VEL
LIN {X 0,Y 392.584,Z 558.533,A -85,B 0,C 180,E1 -11587.918,E2 -11587.918} C_VEL
LIN {X 0,Y 391.953,Z 567.833,A -85,B 0,C 180,E1 -11589.709,E2 -11589.709} C_VEL
LIN {X 0,Y 396.387,Z 599.433,A -85,B 0,C 180,E1 -11590.549,E2 -11590.549} C_VEL
LIN {X 0,Y 395.235,Z 676.9,A -85,B 0,C 180,E1 -11592.037,E2 -11592.037} C_VEL
LIN {X 0,Y 394.603,Z 690.587,A -85,B 0,C 180,E1 -11592.51,E2 -11592.51} C_VEL
LIN {X 0,Y 393.898,Z 702.98,A -85,B 0,C 180,E1 -11593.146,E2 -11593.146} C_VEL
LIN {X 0,Y 392.953,Z 715.672,A -85,B 0,C 180,E1 -11594.039,E2 -11594.039} C_VEL
LIN {X 0,Y 392.092,Z 726.992,A -85,B 0,C 180,E1 -11595.069,E2 -11595.069} C_VEL
LIN {X 0,Y 391.24,Z 737.939,A -85,B 0,C 180,E1 -11596.331,E2 -11596.331} C_VEL
LIN {X 0,Y 390.412,Z 748.046,A -85,B 0,C 180,E1 -11597.789,E2 -11597.789} C_VEL
LIN {X 0,Y 389.651,Z 756.675,A -85,B 0,C 180,E1 -11599.346,E2 -11599.346} C_VEL
LIN {X 0,Y 389.216,Z 763.591,A -85,B 0,C 180,E1 -11600.91,E2 -11600.91} C_VEL
LIN {X 0,Y 388.932,Z 769.941,A -85,B 0,C 180,E1 -11602.733,E2 -11602.733} C_VEL
LIN {X 0,Y 388.787,Z 773.757,A -85,B 0,C 180,E1 -11604.166,E2 -11604.166} C_VEL
LIN {X 0,Y 388.736,Z 777.115,A -85,B 0,C 180,E1 -11605.853,E2 -11605.853} C_VEL
LIN {X 0,Y 388.754,Z 778.605,A -85,B 0,C 180,E1 -11606.891,E2 -11606.891} C_VEL
LIN {X 0,Y 388.846,Z 779.645,A -85,B 0,C 180,E1 -11607.928,E2 -11607.928} C_VEL
LIN {X 0,Y 388.802,Z 780.279,A -85,B 0,C 180,E1 -11608.964,E2 -11608.964} C_VEL
LIN {X 0,Y 388.789,Z 780.518,A -85,B 0,C 180,E1 -11610,E2 -11610} C_VEL
LIN {X 0,Y 388.802,Z 780.339,A -85,B 0,C 180,E1 -11611.036,E2 -11611.036} C_VEL
LIN {X 0,Y 388.843,Z 779.729,A -85,B 0,C 180,E1 -11612.072,E2 -11612.072} C_VEL
LIN {X 0,Y 388.732,Z 777.299,A -85,B 0,C 180,E1 -11614.147,E2 -11614.147} C_VEL
LIN {X 0,Y 388.74,Z 774.19,A -85,B 0,C 180,E1 -11615.77,E2 -11615.77} C_VEL
LIN {X 0,Y 388.931,Z 770.31,A -85,B 0,C 180,E1 -11617.267,E2 -11617.267} C_VEL
LIN {X 0,Y 389.223,Z 764.154,A -85,B 0,C 180,E1 -11619.09,E2 -11619.09} C_VEL
LIN {X 0,Y 389.669,Z 757.413,A -85,B 0,C 180,E1 -11620.653,E2 -11620.653} C_VEL
LIN {X 0,Y 390.431,Z 749.068,A -85,B 0,C 180,E1 -11622.21,E2 -11622.21} C_VEL
LIN {X 0,Y 391.172,Z 740.55,A -85,B 0,C 180,E1 -11623.507,E2 -11623.507} C_VEL
LIN {X 0,Y 392.104,Z 730.079,A -85,B 0,C 180,E1 -11624.798,E2 -11624.798} C_VEL
LIN {X 0,Y 393.072,Z 718.315,A -85,B 0,C 180,E1 -11625.956,E2 -11625.956} C_VEL
LIN {X 0,Y 394.009,Z 706.656,A -85,B 0,C 180,E1 -11626.849,E2 -11626.849} C_VEL
LIN {X 0,Y 394.821,Z 694.608,A -85,B 0,C 180,E1 -11627.547,E2 -11627.547} C_VEL
LIN {X 0,Y 395.575,Z 681.644,A -85,B 0,C 180,E1 -11628.08,E2 -11628.08} C_VEL
LIN {X 0,Y 396.056,Z 667.938,A -85,B 0,C 180,E1 -11628.426,E2 -11628.426} C_VEL
LIN {X 0,Y 396.942,Z 598.382,A -85,B 0,C 180,E1 -11629.763,E2 -11629.763} C_VEL
LIN {X 0,Y 393.505,Z 574.491,A -85,B 0,C 180,E1 -11630.442,E2 -11630.442} C_VEL
LIN {X 0,Y 392.141,Z 566.096,A -85,B 0,C 180,E1 -11630.702,E2 -11630.702} C_VEL
LIN {X 0,Y 393.675,Z 547.548,A -85,B 0,C 180,E1 -11634.429,E2 -11634.429} C_VEL
LIN {X 0,Y 394.154,Z 540.367,A -85,B 0,C 180,E1 -11635.902,E2 -11635.902} C_VEL
LIN {X 0,Y 392.132,Z 529.754,A -85,B 0,C 180,E1 -11638.318,E2 -11638.318} C_VEL
LIN {X 0,Y 390.073,Z 520.898,A -85,B 0,C 180,E1 -11640.446,E2 -11640.446} C_VEL
LIN {X 0,Y 390.068,Z 520.902,A -85,B 0,C 180,E1 -11644.024,E2 -11644.024} C_VEL
LIN {X 0,Y 390.046,Z 520.899,A -85,B 0,C 180,E1 -11647.551,E2 -11647.551} C_VEL
LIN {X 0,Y 390.081,Z 520.895,A -85,B 0,C 180,E1 -11650.825,E2 -11650.825} C_VEL
LIN {X 0,Y 390.1,Z 520.891,A -85,B 0,C 180,E1 -11653.892,E2 -11653.892} C_VEL
LIN {X 0,Y 390.041,Z 520.894,A -85,B 0,C 180,E1 -11657.625,E2 -11657.625} C_VEL
LIN {X 0,Y 390.088,Z 520.894,A -85,B 0,C 180,E1 -11660.907,E2 -11660.907} C_VEL
LIN {X 0,Y 390.081,Z 520.896,A -85,B 0,C 180,E1 -11664.792,E2 -11664.792} C_VEL
LIN {X 0,Y 390.023,Z 520.902,A -85,B 0,C 180,E1 -11668.495,E2 -11668.495} C_VEL
LIN {X 0,Y 390.112,Z 520.887,A -85,B 0,C 180,E1 -11672.069,E2 -11672.069} C_VEL
LIN {X 0,Y 390.073,Z 520.889,A -85,B 0,C 180,E1 -11675.518,E2 -11675.518} C_VEL
LIN {X 0,Y 390.049,Z 520.896,A -85,B 0,C 180,E1 -11678.877,E2 -11678.877} C_VEL
LIN {X 0,Y 390.121,Z 520.887,A -85,B 0,C 180,E1 -11682.166,E2 -11682.166} C_VEL
LIN {X 0,Y 390.138,Z 520.885,A -85,B 0,C 180,E1 -11685.392,E2 -11685.392} C_VEL
LIN {X 0,Y 390.141,Z 520.887,A -85,B 0,C 180,E1 -11688.57,E2 -11688.57} C_VEL
LIN {X 0,Y 390.3,Z 520.865,A -85,B 0,C 180,E1 -11692.031,E2 -11692.031} C_VEL
LIN {X 0,Y 390.226,Z 520.875,A -85,B 0,C 180,E1 -11694.833,E2 -11694.833} C_VEL
LIN {X 0,Y 390.412,Z 520.85,A -85,B 0,C 180,E1 -11697.936,E2 -11697.936} C_VEL
LIN {X 0,Y 390.543,Z 520.833,A -85,B 0,C 180,E1 -11699.999,E2 -11699.999} C_VEL
LIN {X 0,Y 390.309,Z 520.865,A -85,B 0,C 180,E1 -11703.096,E2 -11703.096} C_VEL
LIN {X 0,Y 390.302,Z 520.864,A -85,B 0,C 180,E1 -11706.595,E2 -11706.595} C_VEL
LIN {X 0,Y 390.196,Z 520.88,A -85,B 0,C 180,E1 -11709.328,E2 -11709.328} C_VEL
LIN {X 0,Y 390.162,Z 520.884,A -85,B 0,C 180,E1 -11712.483,E2 -11712.483} C_VEL
LIN {X 0,Y 390.131,Z 520.888,A -85,B 0,C 180,E1 -11715.677,E2 -11715.677} C_VEL
LIN {X 0,Y 390.096,Z 520.895,A -85,B 0,C 180,E1 -11718.922,E2 -11718.922} C_VEL
LIN {X 0,Y 390.03,Z 520.902,A -85,B 0,C 180,E1 -11722.234,E2 -11722.234} C_VEL
LIN {X 0,Y 390.11,Z 520.899,A -85,B 0,C 180,E1 -11725.743,E2 -11725.743} C_VEL
LIN {X 0,Y 390.067,Z 520.9,A -85,B 0,C 180,E1 -11729.108,E2 -11729.108} C_VEL
LIN {X 0,Y 390.11,Z 521.065,A -85,B 0,C 180,E1 -11729.475,E2 -11729.475} C_VEL
LIN {X 0,Y 391.407,Z 527.264,A -85,B 0,C 180,E1 -11731.338,E2 -11731.338} C_VEL
LIN {X 0,Y 396.334,Z 540.56,A -85,B 0,C 180,E1 -11731.914,E2 -11731.914} C_VEL
LIN {X 0,Y 397.743,Z 546.623,A -85,B 0,C 180,E1 -11732.12,E2 -11732.12} C_VEL
LIN {X 0,Y 396.232,Z 633.705,A -85,B 0,C 180,E1 -11733.813,E2 -11733.813} C_VEL
LIN {X 0,Y 395.743,Z 647.499,A -85,B 0,C 180,E1 -11734.303,E2 -11734.303} C_VEL
LIN {X 0,Y 395.208,Z 660.183,A -85,B 0,C 180,E1 -11734.98,E2 -11734.98} C_VEL
LIN {X 0,Y 394.484,Z 671.276,A -85,B 0,C 180,E1 -11735.768,E2 -11735.768} C_VEL
LIN {X 0,Y 393.606,Z 682.924,A -85,B 0,C 180,E1 -11736.831,E2 -11736.831} C_VEL
LIN {X 0,Y 392.674,Z 693.51,A -85,B 0,C 180,E1 -11738.049,E2 -11738.049} C_VEL
LIN {X 0,Y 391.765,Z 703.034,A -85,B 0,C 180,E1 -11739.422,E2 -11739.422} C_VEL
LIN {X 0,Y 390.93,Z 711.694,A -85,B 0,C 180,E1 -11740.971,E2 -11740.971} C_VEL
LIN {X 0,Y 390.281,Z 718.185,A -85,B 0,C 180,E1 -11742.414,E2 -11742.414} C_VEL
LIN {X 0,Y 389.775,Z 723.405,A -85,B 0,C 180,E1 -11743.845,E2 -11743.845} C_VEL
LIN {X 0,Y 389.456,Z 727.556,A -85,B 0,C 180,E1 -11745.27,E2 -11745.27} C_VEL
LIN {X 0,Y 389.167,Z 730.74,A -85,B 0,C 180,E1 -11746.668,E2 -11746.668} C_VEL
LIN {X 0,Y 388.956,Z 733.098,A -85,B 0,C 180,E1 -11748.046,E2 -11748.046} C_VEL
LIN {X 0,Y 388.763,Z 734.703,A -85,B 0,C 180,E1 -11749.399,E2 -11749.399} C_VEL
LIN {X 0,Y 388.638,Z 735.697,A -85,B 0,C 180,E1 -11751.04,E2 -11751.04} C_VEL
LIN {X 0,Y 388.628,Z 735.68,A -85,B 0,C 180,E1 -11752.721,E2 -11752.721} C_VEL
LIN {X 0,Y 388.753,Z 734.341,A -85,B 0,C 180,E1 -11754.655,E2 -11754.655} C_VEL
LIN {X 0,Y 388.917,Z 732.23,A -85,B 0,C 180,E1 -11756.227,E2 -11756.227} C_VEL
LIN {X 0,Y 389.22,Z 728.483,A -85,B 0,C 180,E1 -11758.065,E2 -11758.065} C_VEL
LIN {X 0,Y 389.658,Z 723.07,A -85,B 0,C 180,E1 -11759.966,E2 -11759.966} C_VEL
LIN {X 0,Y 390.216,Z 716.344,A -85,B 0,C 180,E1 -11761.732,E2 -11761.732} C_VEL
LIN {X 0,Y 390.855,Z 708.866,A -85,B 0,C 180,E1 -11763.287,E2 -11763.287} C_VEL
LIN {X 0,Y 391.646,Z 699.961,A -85,B 0,C 180,E1 -11764.775,E2 -11764.775} C_VEL
LIN {X 0,Y 392.431,Z 690.132,A -85,B 0,C 180,E1 -11766.093,E2 -11766.093} C_VEL
LIN {X 0,Y 393.232,Z 679.303,A -85,B 0,C 180,E1 -11767.264,E2 -11767.264} C_VEL
LIN {X 0,Y 394.06,Z 667.279,A -85,B 0,C 180,E1 -11768.28,E2 -11768.28} C_VEL
LIN {X 0,Y 394.719,Z 655.061,A -85,B 0,C 180,E1 -11769.071,E2 -11769.071} C_VEL
LIN {X 0,Y 395.262,Z 642.235,A -85,B 0,C 180,E1 -11769.675,E2 -11769.675} C_VEL
LIN {X 0,Y 395.564,Z 628.782,A -85,B 0,C 180,E1 -11770.078,E2 -11770.078} C_VEL
LIN {X 0,Y 396.819,Z 545.914,A -85,B 0,C 180,E1 -11771.65,E2 -11771.65} C_VEL
LIN {X 0,Y 394.329,Z 535.546,A -85,B 0,C 180,E1 -11771.978,E2 -11771.978} C_VEL
LIN {X 0,Y 391.055,Z 525.693,A -85,B 0,C 180,E1 -11772.346,E2 -11772.346} C_VEL
LIN {X 0,Y 390.133,Z 520.888,A -85,B 0,C 180,E1 -11773.719,E2 -11773.719} C_VEL
LIN {X 0,Y 390.164,Z 520.881,A -85,B 0,C 180,E1 -11777.373,E2 -11777.373} C_VEL
LIN {X 0,Y 390.202,Z 520.88,A -85,B 0,C 180,E1 -11780.671,E2 -11780.671} C_VEL
LIN {X 0,Y 390.285,Z 520.865,A -85,B 0,C 180,E1 -11781.853,E2 -11781.853} C_VEL
LIN {X 0,Y 389.644,Z 520.95,A -85,B 0,C 180,E1 -11782.715,E2 -11782.715} C_VEL
LIN {X 0,Y 386.68,Z 521.315,A -85,B 0,C 180,E1 -11784.113,E2 -11784.113} C_VEL
LIN {X 0,Y 384.191,Z 521.628,A -85,B 0,C 180,E1 -11785.244,E2 -11785.244} C_VEL
LIN {X 0,Y 383.199,Z 521.749,A -85,B 0,C 180,E1 -11786.12,E2 -11786.12} C_VEL
LIN {X 0,Y 383.161,Z 521.755,A -85,B 0,C 180,E1 -11786.417,E2 -11786.417} C_VEL
LIN {X 0,Y 383.385,Z 521.725,A -85,B 0,C 180,E1 -11787.899,E2 -11787.899} C_VEL
LIN {X 0,Y 383.517,Z 521.708,A -85,B 0,C 180,E1 -11790,E2 -11790} C_VEL
LIN {X 0,Y 383.249,Z 521.746,A -85,B 0,C 180,E1 -11793.154,E2 -11793.154} C_VEL
LIN {X 0,Y 383.285,Z 521.738,A -85,B 0,C 180,E1 -11796.316,E2 -11796.316} C_VEL
LIN {X 0,Y 383.257,Z 521.743,A -85,B 0,C 180,E1 -11798.436,E2 -11798.436} C_VEL
LIN {X 0,Y 383.094,Z 521.762,A -85,B 0,C 180,E1 -11801.642,E2 -11801.642} C_VEL
LIN {X 0,Y 383.107,Z 521.766,A -85,B 0,C 180,E1 -11804.881,E2 -11804.881} C_VEL
LIN {X 0,Y 383.059,Z 521.766,A -85,B 0,C 180,E1 -11808.173,E2 -11808.173} C_VEL
LIN {X 0,Y 382.989,Z 521.776,A -85,B 0,C 180,E1 -11811.531,E2 -11811.531} C_VEL
LIN {X 0,Y 383.048,Z 521.774,A -85,B 0,C 180,E1 -11814.96,E2 -11814.96} C_VEL
LIN {X 0,Y 383.045,Z 521.769,A -85,B 0,C 180,E1 -11818.492,E2 -11818.492} C_VEL
LIN {X 0,Y 383.032,Z 521.769,A -85,B 0,C 180,E1 -11822.147,E2 -11822.147} C_VEL
LIN {X 0,Y 383.021,Z 521.77,A -85,B 0,C 180,E1 -11825.955,E2 -11825.955} C_VEL
LIN {X 0,Y 383.016,Z 521.772,A -85,B 0,C 180,E1 -11829.588,E2 -11829.588} C_VEL
LIN {X 0,Y 383.058,Z 521.769,A -85,B 0,C 180,E1 -11832.788,E2 -11832.788} C_VEL
LIN {X 0,Y 383.062,Z 521.766,A -85,B 0,C 180,E1 -11835.799,E2 -11835.799} C_VEL
LIN {X 0,Y 383.037,Z 521.772,A -85,B 0,C 180,E1 -11838.786,E2 -11838.786} C_VEL
LIN {X 0,Y 382.996,Z 521.773,A -85,B 0,C 180,E1 -11842.095,E2 -11842.095} C_VEL
LIN {X 0,Y 383.01,Z 521.776,A -85,B 0,C 180,E1 -11845.332,E2 -11845.332} C_VEL
LIN {X 0,Y 382.978,Z 521.782,A -85,B 0,C 180,E1 -11849.082,E2 -11849.082} C_VEL
LIN {X 0,Y 383.048,Z 521.769,A -85,B 0,C 180,E1 -11852.698,E2 -11852.698} C_VEL
LIN {X 0,Y 383.042,Z 521.774,A -85,B 0,C 180,E1 -11855.04,E2 -11855.04} C_VEL
LIN {X 0,Y 382.983,Z 521.776,A -85,B 0,C 180,E1 -11858.469,E2 -11858.469} C_VEL
LIN {X 0,Y 383.054,Z 521.767,A -85,B 0,C 180,E1 -11861.827,E2 -11861.827} C_VEL
LIN {X 0,Y 383.102,Z 521.767,A -85,B 0,C 180,E1 -11865.119,E2 -11865.119} C_VEL
LIN {X 0,Y 383.099,Z 521.761,A -85,B 0,C 180,E1 -11868.359,E2 -11868.359} C_VEL
LIN {X 0,Y 383.295,Z 521.736,A -85,B 0,C 180,E1 -11871.933,E2 -11871.933} C_VEL
LIN {X 0,Y 383.198,Z 521.75,A -85,B 0,C 180,E1 -11874.739,E2 -11874.739} C_VEL
LIN {X 0,Y 383.38,Z 521.726,A -85,B 0,C 180,E1 -11877.899,E2 -11877.899} C_VEL
LIN {X 0,Y 383.513,Z 521.709,A -85,B 0,C 180,E1 -11880.001,E2 -11880.001} C_VEL
LIN {X 0,Y 383.275,Z 521.745,A -85,B 0,C 180,E1 -11883.154,E2 -11883.154} C_VEL
LIN {X 0,Y 383.284,Z 521.737,A -85,B 0,C 180,E1 -11886.317,E2 -11886.317} C_VEL
LIN {X 0,Y 383.144,Z 521.759,A -85,B 0,C 180,E1 -11889.503,E2 -11889.503} C_VEL
LIN {X 0,Y 383.118,Z 521.762,A -85,B 0,C 180,E1 -11893.537,E2 -11893.537} C_VEL
LIN {X 0,Y 383.088,Z 521.767,A -85,B 0,C 180,E1 -11897.455,E2 -11897.455} C_VEL
LIN {X 0,Y 383.022,Z 521.771,A -85,B 0,C 180,E1 -11900.648,E2 -11900.648} C_VEL
LIN {X 0,Y 383.027,Z 521.771,A -85,B 0,C 180,E1 -11903.808,E2 -11903.808} C_VEL
LIN {X 0,Y 383.074,Z 521.764,A -85,B 0,C 180,E1 -11906.124,E2 -11906.124} C_VEL
LIN {X 0,Y 383.044,Z 521.768,A -85,B 0,C 180,E1 -11908.493,E2 -11908.493} C_VEL
LIN {X 0,Y 383.004,Z 521.772,A -85,B 0,C 180,E1 -11912.428,E2 -11912.428} C_VEL
LIN {X 0,Y 383.029,Z 521.769,A -85,B 0,C 180,E1 -11916.166,E2 -11916.166} C_VEL
LIN {X 0,Y 383.006,Z 521.773,A -85,B 0,C 180,E1 -11919.959,E2 -11919.959} C_VEL
LIN {X 0,Y 383.002,Z 521.774,A -85,B 0,C 180,E1 -11922.78,E2 -11922.78} C_VEL
LIN {X 0,Y 383.036,Z 521.771,A -85,B 0,C 180,E1 -11925.796,E2 -11925.796} C_VEL
LIN {X 0,Y 383.043,Z 521.769,A -85,B 0,C 180,E1 -11928.787,E2 -11928.787} C_VEL
LIN {X 0,Y 383.002,Z 521.773,A -85,B 0,C 180,E1 -11932.097,E2 -11932.097} C_VEL
LIN {X 0,Y 383.018,Z 521.777,A -85,B 0,C 180,E1 -11935.333,E2 -11935.333} C_VEL
LIN {X 0,Y 382.983,Z 521.779,A -85,B 0,C 180,E1 -11939.082,E2 -11939.082} C_VEL
LIN {X 0,Y 383.042,Z 521.969,A -85,B 0,C 180,E1 -11939.696,E2 -11939.696} C_VEL
LIN {X 0,Y 386.115,Z 536.035,A -85,B 0,C 180,E1 -11942.933,E2 -11942.933} C_VEL
LIN {X 0,Y 387.061,Z 541.618,A -85,B 0,C 180,E1 -11944.166,E2 -11944.166} C_VEL
LIN {X 0,Y 385.821,Z 556.649,A -85,B 0,C 180,E1 -11947.227,E2 -11947.227} C_VEL
LIN {X 0,Y 384.999,Z 567.131,A -85,B 0,C 180,E1 -11949.34,E2 -11949.34} C_VEL
LIN {X 0,Y 389.608,Z 599.611,A -85,B 0,C 180,E1 -11950.234,E2 -11950.234} C_VEL
LIN {X 0,Y 388.435,Z 676.672,A -85,B 0,C 180,E1 -11951.746,E2 -11951.746} C_VEL
LIN {X 0,Y 387.756,Z 690.292,A -85,B 0,C 180,E1 -11952.225,E2 -11952.225} C_VEL
LIN {X 0,Y 387.048,Z 702.111,A -85,B 0,C 180,E1 -11952.839,E2 -11952.839} C_VEL
LIN {X 0,Y 386.257,Z 713.346,A -85,B 0,C 180,E1 -11953.619,E2 -11953.619} C_VEL
LIN {X 0,Y 385.265,Z 725.009,A -85,B 0,C 180,E1 -11954.663,E2 -11954.663} C_VEL
LIN {X 0,Y 384.444,Z 735.404,A -85,B 0,C 180,E1 -11955.832,E2 -11955.832} C_VEL
LIN {X 0,Y 383.668,Z 744.132,A -85,B 0,C 180,E1 -11957.033,E2 -11957.033} C_VEL
LIN {X 0,Y 383.002,Z 752.066,A -85,B 0,C 180,E1 -11958.355,E2 -11958.355} C_VEL
LIN {X 0,Y 382.4,Z 759.804,A -85,B 0,C 180,E1 -11959.945,E2 -11959.945} C_VEL
LIN {X 0,Y 382.01,Z 766.021,A -85,B 0,C 180,E1 -11961.537,E2 -11961.537} C_VEL
LIN {X 0,Y 381.836,Z 770.951,A -85,B 0,C 180,E1 -11963.129,E2 -11963.129} C_VEL
LIN {X 0,Y 381.703,Z 774.725,A -85,B 0,C 180,E1 -11964.718,E2 -11964.718} C_VEL
LIN {X 0,Y 381.662,Z 776.667,A -85,B 0,C 180,E1 -11965.776,E2 -11965.776} C_VEL
LIN {X 0,Y 381.658,Z 778.17,A -85,B 0,C 180,E1 -11966.833,E2 -11966.833} C_VEL
LIN {X 0,Y 381.776,Z 779.221,A -85,B 0,C 180,E1 -11967.89,E2 -11967.89} C_VEL
LIN {X 0,Y 381.732,Z 779.861,A -85,B 0,C 180,E1 -11968.945,E2 -11968.945} C_VEL
LIN {X 0,Y 381.717,Z 780.105,A -85,B 0,C 180,E1 -11970,E2 -11970} C_VEL
LIN {X 0,Y 381.732,Z 779.938,A -85,B 0,C 180,E1 -11971.055,E2 -11971.055} C_VEL
LIN {X 0,Y 381.754,Z 779.333,A -85,B 0,C 180,E1 -11972.11,E2 -11972.11} C_VEL
LIN {X 0,Y 381.655,Z 776.912,A -85,B 0,C 180,E1 -11974.224,E2 -11974.224} C_VEL
LIN {X 0,Y 381.694,Z 773.251,A -85,B 0,C 180,E1 -11976.125,E2 -11976.125} C_VEL
LIN {X 0,Y 381.906,Z 768.343,A -85,B 0,C 180,E1 -11977.933,E2 -11977.933} C_VEL
LIN {X 0,Y 382.335,Z 761.737,A -85,B 0,C 180,E1 -11979.789,E2 -11979.789} C_VEL
LIN {X 0,Y 382.877,Z 754.523,A -85,B 0,C 180,E1 -11981.38,E2 -11981.38} C_VEL
LIN {X 0,Y 383.782,Z 745.553,A -85,B 0,C 180,E1 -11982.963,E2 -11982.963} C_VEL
LIN {X 0,Y 384.583,Z 736.711,A -85,B 0,C 180,E1 -11984.237,E2 -11984.237} C_VEL
LIN {X 0,Y 385.53,Z 726.283,A -85,B 0,C 180,E1 -11985.462,E2 -11985.462} C_VEL
LIN {X 0,Y 386.497,Z 715.094,A -85,B 0,C 180,E1 -11986.506,E2 -11986.506} C_VEL
LIN {X 0,Y 387.471,Z 702.601,A -85,B 0,C 180,E1 -11987.414,E2 -11987.414} C_VEL
LIN {X 0,Y 388.313,Z 689.988,A -85,B 0,C 180,E1 -11988.089,E2 -11988.089} C_VEL
LIN {X 0,Y 389.111,Z 676.763,A -85,B 0,C 180,E1 -11988.562,E2 -11988.562} C_VEL
LIN {X 0,Y 389.591,Z 650.166,A -85,B 0,C 180,E1 -11989.117,E2 -11989.117} C_VEL
LIN {X 0,Y 390.335,Z 599.392,A -85,B 0,C 180,E1 -11990.112,E2 -11990.112} C_VEL
LIN {X 0,Y 387.137,Z 576.888,A -85,B 0,C 180,E1 -11990.77,E2 -11990.77} C_VEL
LIN {X 0,Y 385.282,Z 565.649,A -85,B 0,C 180,E1 -11991.127,E2 -11991.127} C_VEL
LIN {X 0,Y 386.935,Z 547.008,A -85,B 0,C 180,E1 -11994.95,E2 -11994.95} C_VEL
LIN {X 0,Y 387.234,Z 541.513,A -85,B 0,C 180,E1 -11996.111,E2 -11996.111} C_VEL
LIN {X 0,Y 385.167,Z 530.887,A -85,B 0,C 180,E1 -11998.591,E2 -11998.591} C_VEL
LIN {X 0,Y 383.004,Z 521.779,A -85,B 0,C 180,E1 -12000.842,E2 -12000.842} C_VEL
LIN {X 0,Y 383.018,Z 521.78,A -85,B 0,C 180,E1 -12004.667,E2 -12004.667} C_VEL
LIN {X 0,Y 383.002,Z 521.777,A -85,B 0,C 180,E1 -12007.903,E2 -12007.903} C_VEL
LIN {X 0,Y 383.045,Z 521.771,A -85,B 0,C 180,E1 -12011.338,E2 -12011.338} C_VEL
LIN {X 0,Y 383.033,Z 521.774,A -85,B 0,C 180,E1 -12014.308,E2 -12014.308} C_VEL
LIN {X 0,Y 383.007,Z 521.772,A -85,B 0,C 180,E1 -12017.239,E2 -12017.239} C_VEL
LIN {X 0,Y 383.012,Z 521.773,A -85,B 0,C 180,E1 -12020.412,E2 -12020.412} C_VEL
LIN {X 0,Y 383.022,Z 521.771,A -85,B 0,C 180,E1 -12024.044,E2 -12024.044} C_VEL
LIN {X 0,Y 382.983,Z 521.777,A -85,B 0,C 180,E1 -12027.577,E2 -12027.577} C_VEL
LIN {X 0,Y 382.993,Z 521.776,A -85,B 0,C 180,E1 -12030.3,E2 -12030.3} C_VEL
LIN {X 0,Y 383.051,Z 521.768,A -85,B 0,C 180,E1 -12032.697,E2 -12032.697} C_VEL
LIN {X 0,Y 383.046,Z 521.767,A -85,B 0,C 180,E1 -12035.039,E2 -12035.039} C_VEL
LIN {X 0,Y 382.986,Z 521.778,A -85,B 0,C 180,E1 -12038.468,E2 -12038.468} C_VEL
LIN {X 0,Y 383.056,Z 521.766,A -85,B 0,C 180,E1 -12041.826,E2 -12041.826} C_VEL
LIN {X 0,Y 383.104,Z 521.764,A -85,B 0,C 180,E1 -12045.118,E2 -12045.118} C_VEL
LIN {X 0,Y 383.091,Z 521.764,A -85,B 0,C 180,E1 -12048.357,E2 -12048.357} C_VEL
LIN {X 0,Y 383.256,Z 521.742,A -85,B 0,C 180,E1 -12051.974,E2 -12051.974} C_VEL
LIN {X 0,Y 383.198,Z 521.749,A -85,B 0,C 180,E1 -12054.738,E2 -12054.738} C_VEL
LIN {X 0,Y 383.38,Z 521.726,A -85,B 0,C 180,E1 -12057.898,E2 -12057.898} C_VEL
LIN {X 0,Y 383.513,Z 521.708,A -85,B 0,C 180,E1 -12059.999,E2 -12059.999} C_VEL
LIN {X 0,Y 383.246,Z 521.744,A -85,B 0,C 180,E1 -12063.153,E2 -12063.153} C_VEL
LIN {X 0,Y 383.262,Z 521.74,A -85,B 0,C 180,E1 -12066.585,E2 -12066.585} C_VEL
LIN {X 0,Y 383.143,Z 521.76,A -85,B 0,C 180,E1 -12069.502,E2 -12069.502} C_VEL
LIN {X 0,Y 383.116,Z 521.762,A -85,B 0,C 180,E1 -12073.536,E2 -12073.536} C_VEL
LIN {X 0,Y 383.085,Z 521.767,A -85,B 0,C 180,E1 -12077.454,E2 -12077.454} C_VEL
LIN {X 0,Y 383.02,Z 521.775,A -85,B 0,C 180,E1 -12080.647,E2 -12080.647} C_VEL
LIN {X 0,Y 383.025,Z 521.779,A -85,B 0,C 180,E1 -12083.807,E2 -12083.807} C_VEL
LIN {X 0,Y 383.071,Z 521.775,A -85,B 0,C 180,E1 -12086.123,E2 -12086.123} C_VEL
LIN {X 0,Y 383.044,Z 521.871,A -85,B 0,C 180,E1 -12089.091,E2 -12089.091} C_VEL
LIN {X 0,Y 384.278,Z 527.673,A -85,B 0,C 180,E1 -12090.878,E2 -12090.878} C_VEL
LIN {X 0,Y 389.882,Z 542.307,A -85,B 0,C 180,E1 -12091.558,E2 -12091.558} C_VEL
LIN {X 0,Y 391.185,Z 548.764,A -85,B 0,C 180,E1 -12091.773,E2 -12091.773} C_VEL
LIN {X 0,Y 389.561,Z 633.961,A -85,B 0,C 180,E1 -12093.46,E2 -12093.46} C_VEL
LIN {X 0,Y 389.048,Z 647.844,A -85,B 0,C 180,E1 -12093.96,E2 -12093.96} C_VEL
LIN {X 0,Y 388.487,Z 660.741,A -85,B 0,C 180,E1 -12094.661,E2 -12094.661} C_VEL
LIN {X 0,Y 387.65,Z 672.745,A -85,B 0,C 180,E1 -12095.54,E2 -12095.54} C_VEL
LIN {X 0,Y 386.741,Z 684.399,A -85,B 0,C 180,E1 -12096.642,E2 -12096.642} C_VEL
LIN {X 0,Y 385.836,Z 693.906,A -85,B 0,C 180,E1 -12097.768,E2 -12097.768} C_VEL
LIN {X 0,Y 384.838,Z 703.784,A -85,B 0,C 180,E1 -12099.221,E2 -12099.221} C_VEL
LIN {X 0,Y 384.064,Z 711.342,A -85,B 0,C 180,E1 -12100.59,E2 -12100.59} C_VEL
LIN {X 0,Y 383.354,Z 717.979,A -85,B 0,C 180,E1 -12102.059,E2 -12102.059} C_VEL
LIN {X 0,Y 382.724,Z 724.488,A -85,B 0,C 180,E1 -12103.885,E2 -12103.885} C_VEL
LIN {X 0,Y 382.254,Z 729.617,A -85,B 0,C 180,E1 -12105.81,E2 -12105.81} C_VEL
LIN {X 0,Y 381.966,Z 732.663,A -85,B 0,C 180,E1 -12107.389,E2 -12107.389} C_VEL
LIN {X 0,Y 381.715,Z 734.794,A -85,B 0,C 180,E1 -12109.014,E2 -12109.014} C_VEL
LIN {X 0,Y 381.557,Z 735.974,A -85,B 0,C 180,E1 -12110.678,E2 -12110.678} C_VEL
LIN {X 0,Y 381.563,Z 736.116,A -85,B 0,C 180,E1 -12112.569,E2 -12112.569} C_VEL
LIN {X 0,Y 381.605,Z 735.257,A -85,B 0,C 180,E1 -12114.129,E2 -12114.129} C_VEL
LIN {X 0,Y 381.796,Z 733.183,A -85,B 0,C 180,E1 -12115.928,E2 -12115.928} C_VEL
LIN {X 0,Y 382.084,Z 729.743,A -85,B 0,C 180,E1 -12117.791,E2 -12117.791} C_VEL
LIN {X 0,Y 382.523,Z 724.631,A -85,B 0,C 180,E1 -12119.713,E2 -12119.713} C_VEL
LIN {X 0,Y 383.072,Z 718.305,A -85,B 0,C 180,E1 -12121.511,E2 -12121.511} C_VEL
LIN {X 0,Y 383.646,Z 711.612,A -85,B 0,C 180,E1 -12123.012,E2 -12123.012} C_VEL
LIN {X 0,Y 384.41,Z 703.048,A -85,B 0,C 180,E1 -12124.556,E2 -12124.556} C_VEL
LIN {X 0,Y 385.316,Z 693.223,A -85,B 0,C 180,E1 -12125.984,E2 -12125.984} C_VEL
LIN {X 0,Y 386.054,Z 683.751,A -85,B 0,C 180,E1 -12127.1,E2 -12127.1} C_VEL
LIN {X 0,Y 386.888,Z 672.658,A -85,B 0,C 180,E1 -12128.148,E2 -12128.148} C_VEL
LIN {X 0,Y 387.6,Z 660.951,A -85,B 0,C 180,E1 -12129.016,E2 -12129.016} C_VEL
LIN {X 0,Y 388.179,Z 649.294,A -85,B 0,C 180,E1 -12129.673,E2 -12129.673} C_VEL
LIN {X 0,Y 388.65,Z 636.1,A -85,B 0,C 180,E1 -12130.189,E2 -12130.189} C_VEL
LIN {X 0,Y 388.984,Z 619.039,A -85,B 0,C 180,E1 -12130.574,E2 -12130.574} C_VEL
LIN {X 0,Y 390.117,Z 546.817,A -85,B 0,C 180,E1 -12131.963,E2 -12131.963} C_VEL
LIN {X 0,Y 387.61,Z 536.834,A -85,B 0,C 180,E1 -12132.293,E2 -12132.293} C_VEL
LIN {X 0,Y 383.913,Z 525.949,A -85,B 0,C 180,E1 -12132.738,E2 -12132.738} C_VEL
LIN {X 0,Y 383.119,Z 521.761,A -85,B 0,C 180,E1 -12133.96,E2 -12133.96} C_VEL
LIN {X 0,Y 383.133,Z 521.759,A -85,B 0,C 180,E1 -12137.284,E2 -12137.284} C_VEL
LIN {X 0,Y 383.148,Z 521.757,A -85,B 0,C 180,E1 -12140.498,E2 -12140.498} C_VEL
LIN {X 0,Y 383.277,Z 521.739,A -85,B 0,C 180,E1 -12143.684,E2 -12143.684} C_VEL
LIN {X 0,Y 383.161,Z 521.755,A -85,B 0,C 180,E1 -12146.417,E2 -12146.417} C_VEL
LIN {X 0,Y 382.617,Z 521.829,A -85,B 0,C 180,E1 -12147.295,E2 -12147.295} C_VEL
LIN {X 0,Y 379.832,Z 522.184,A -85,B 0,C 180,E1 -12148.724,E2 -12148.724} C_VEL
LIN {X 0,Y 377.406,Z 522.485,A -85,B 0,C 180,E1 -12149.88,E2 -12149.88} C_VEL
LIN {X 0,Y 376.363,Z 522.608,A -85,B 0,C 180,E1 -12150.773,E2 -12150.773} C_VEL
LIN {X 0,Y 376.281,Z 522.615,A -85,B 0,C 180,E1 -12151.076,E2 -12151.076} C_VEL
LIN {X 0,Y 376.187,Z 522.625,A -85,B 0,C 180,E1 -12153.213,E2 -12153.213} C_VEL
LIN {X 0,Y 376.244,Z 522.616,A -85,B 0,C 180,E1 -12156.435,E2 -12156.435} C_VEL
LIN {X 0,Y 376.202,Z 522.623,A -85,B 0,C 180,E1 -12158.595,E2 -12158.595} C_VEL
LIN {X 0,Y 376.047,Z 522.639,A -85,B 0,C 180,E1 -12161.863,E2 -12161.863} C_VEL
LIN {X 0,Y 376.055,Z 522.643,A -85,B 0,C 180,E1 -12165.167,E2 -12165.167} C_VEL
LIN {X 0,Y 376.005,Z 522.646,A -85,B 0,C 180,E1 -12168.526,E2 -12168.526} C_VEL
LIN {X 0,Y 375.959,Z 522.65,A -85,B 0,C 180,E1 -12171.954,E2 -12171.954} C_VEL
LIN {X 0,Y 376.001,Z 522.647,A -85,B 0,C 180,E1 -12175.461,E2 -12175.461} C_VEL
LIN {X 0,Y 375.972,Z 522.655,A -85,B 0,C 180,E1 -12179.078,E2 -12179.078} C_VEL
LIN {X 0,Y 375.951,Z 522.656,A -85,B 0,C 180,E1 -12182.827,E2 -12182.827} C_VEL
LIN {X 0,Y 375.953,Z 522.654,A -85,B 0,C 180,E1 -12185.415,E2 -12185.415} C_VEL
LIN {X 0,Y 375.972,Z 522.649,A -85,B 0,C 180,E1 -12188.271,E2 -12188.271} C_VEL
LIN {X 0,Y 375.983,Z 522.648,A -85,B 0,C 180,E1 -12191.61,E2 -12191.61} C_VEL
LIN {X 0,Y 376.007,Z 522.649,A -85,B 0,C 180,E1 -12195.255,E2 -12195.255} C_VEL
LIN {X 0,Y 375.993,Z 522.652,A -85,B 0,C 180,E1 -12199.141,E2 -12199.141} C_VEL
LIN {X 0,Y 375.96,Z 522.65,A -85,B 0,C 180,E1 -12201.912,E2 -12201.912} C_VEL
LIN {X 0,Y 375.972,Z 522.653,A -85,B 0,C 180,E1 -12205.333,E2 -12205.333} C_VEL
LIN {X 0,Y 375.951,Z 522.652,A -85,B 0,C 180,E1 -12208.438,E2 -12208.438} C_VEL
LIN {X 0,Y 375.994,Z 522.646,A -85,B 0,C 180,E1 -12212.142,E2 -12212.142} C_VEL
LIN {X 0,Y 375.997,Z 522.646,A -85,B 0,C 180,E1 -12214.539,E2 -12214.539} C_VEL
LIN {X 0,Y 375.949,Z 522.651,A -85,B 0,C 180,E1 -12218.045,E2 -12218.045} C_VEL
LIN {X 0,Y 376,Z 522.648,A -85,B 0,C 180,E1 -12221.473,E2 -12221.473} C_VEL
LIN {X 0,Y 376.05,Z 522.642,A -85,B 0,C 180,E1 -12224.833,E2 -12224.833} C_VEL
LIN {X 0,Y 376.05,Z 522.639,A -85,B 0,C 180,E1 -12228.137,E2 -12228.137} C_VEL
LIN {X 0,Y 376.249,Z 522.614,A -85,B 0,C 180,E1 -12231.878,E2 -12231.878} C_VEL
LIN {X 0,Y 376.17,Z 522.625,A -85,B 0,C 180,E1 -12234.64,E2 -12234.64} C_VEL
LIN {X 0,Y 376.346,Z 522.603,A -85,B 0,C 180,E1 -12237.86,E2 -12237.86} C_VEL
LIN {X 0,Y 376.482,Z 522.585,A -85,B 0,C 180,E1 -12240.001,E2 -12240.001} C_VEL
LIN {X 0,Y 376.212,Z 522.626,A -85,B 0,C 180,E1 -12243.213,E2 -12243.213} C_VEL
LIN {X 0,Y 376.241,Z 522.615,A -85,B 0,C 180,E1 -12246.436,E2 -12246.436} C_VEL
LIN {X 0,Y 376.112,Z 522.633,A -85,B 0,C 180,E1 -12249.682,E2 -12249.682} C_VEL
LIN {X 0,Y 376.082,Z 522.637,A -85,B 0,C 180,E1 -12253.658,E2 -12253.658} C_VEL
LIN {X 0,Y 376.036,Z 522.643,A -85,B 0,C 180,E1 -12257.608,E2 -12257.608} C_VEL
LIN {X 0,Y 375.972,Z 522.651,A -85,B 0,C 180,E1 -12260.833,E2 -12260.833} C_VEL
LIN {X 0,Y 375.988,Z 522.646,A -85,B 0,C 180,E1 -12264.282,E2 -12264.282} C_VEL
LIN {X 0,Y 376.014,Z 522.644,A -85,B 0,C 180,E1 -12266.653,E2 -12266.653} C_VEL
LIN {X 0,Y 375.972,Z 522.653,A -85,B 0,C 180,E1 -12269.08,E2 -12269.08} C_VEL
LIN {X 0,Y 375.952,Z 522.653,A -85,B 0,C 180,E1 -12272.829,E2 -12272.829} C_VEL
LIN {X 0,Y 375.954,Z 522.656,A -85,B 0,C 180,E1 -12275.416,E2 -12275.416} C_VEL
LIN {X 0,Y 375.972,Z 522.648,A -85,B 0,C 180,E1 -12278.272,E2 -12278.272} C_VEL
LIN {X 0,Y 375.933,Z 522.657,A -85,B 0,C 180,E1 -12281.602,E2 -12281.602} C_VEL
LIN {X 0,Y 375.977,Z 522.654,A -85,B 0,C 180,E1 -12285.262,E2 -12285.262} C_VEL
LIN {X 0,Y 375.988,Z 522.646,A -85,B 0,C 180,E1 -12288.391,E2 -12288.391} C_VEL
LIN {X 0,Y 375.967,Z 522.65,A -85,B 0,C 180,E1 -12291.913,E2 -12291.913} C_VEL
LIN {X 0,Y 375.98,Z 522.654,A -85,B 0,C 180,E1 -12295.334,E2 -12295.334} C_VEL
LIN {X 0,Y 375.958,Z 522.655,A -85,B 0,C 180,E1 -12298.439,E2 -12298.439} C_VEL
LIN {X 0,Y 375.947,Z 522.69,A -85,B 0,C 180,E1 -12299.354,E2 -12299.354} C_VEL
LIN {X 0,Y 378.757,Z 535.452,A -85,B 0,C 180,E1 -12302.363,E2 -12302.363} C_VEL
LIN {X 0,Y 380.062,Z 542.449,A -85,B 0,C 180,E1 -12303.949,E2 -12303.949} C_VEL
LIN {X 0,Y 379.449,Z 550.973,A -85,B 0,C 180,E1 -12305.73,E2 -12305.73} C_VEL
LIN {X 0,Y 378.133,Z 566.779,A -85,B 0,C 180,E1 -12308.985,E2 -12308.985} C_VEL
LIN {X 0,Y 382.849,Z 600.691,A -85,B 0,C 180,E1 -12309.931,E2 -12309.931} C_VEL
LIN {X 0,Y 381.631,Z 676.265,A -85,B 0,C 180,E1 -12311.444,E2 -12311.444} C_VEL
LIN {X 0,Y 380.938,Z 689.886,A -85,B 0,C 180,E1 -12311.931,E2 -12311.931} C_VEL
LIN {X 0,Y 380.15,Z 702.248,A -85,B 0,C 180,E1 -12312.587,E2 -12312.587} C_VEL
LIN {X 0,Y 379.285,Z 714.144,A -85,B 0,C 180,E1 -12313.448,E2 -12313.448} C_VEL
LIN {X 0,Y 378.261,Z 725.595,A -85,B 0,C 180,E1 -12314.51,E2 -12314.51} C_VEL
LIN {X 0,Y 377.43,Z 735.754,A -85,B 0,C 180,E1 -12315.691,E2 -12315.691} C_VEL
LIN {X 0,Y 376.547,Z 745.235,A -85,B 0,C 180,E1 -12317.058,E2 -12317.058} C_VEL
LIN {X 0,Y 375.725,Z 754.272,A -85,B 0,C 180,E1 -12318.674,E2 -12318.674} C_VEL
LIN {X 0,Y 375.181,Z 761.544,A -85,B 0,C 180,E1 -12320.294,E2 -12320.294} C_VEL
LIN {X 0,Y 374.85,Z 767.331,A -85,B 0,C 180,E1 -12321.917,E2 -12321.917} C_VEL
LIN {X 0,Y 374.638,Z 772.621,A -85,B 0,C 180,E1 -12323.857,E2 -12323.857} C_VEL
LIN {X 0,Y 374.588,Z 776.219,A -85,B 0,C 180,E1 -12325.696,E2 -12325.696} C_VEL
LIN {X 0,Y 374.564,Z 777.735,A -85,B 0,C 180,E1 -12326.773,E2 -12326.773} C_VEL
LIN {X 0,Y 374.689,Z 778.795,A -85,B 0,C 180,E1 -12327.85,E2 -12327.85} C_VEL
LIN {X 0,Y 374.664,Z 779.442,A -85,B 0,C 180,E1 -12328.925,E2 -12328.925} C_VEL
LIN {X 0,Y 374.647,Z 779.693,A -85,B 0,C 180,E1 -12330,E2 -12330} C_VEL
LIN {X 0,Y 374.663,Z 779.537,A -85,B 0,C 180,E1 -12331.075,E2 -12331.075} C_VEL
LIN {X 0,Y 374.668,Z 778.936,A -85,B 0,C 180,E1 -12332.15,E2 -12332.15} C_VEL
LIN {X 0,Y 374.579,Z 776.528,A -85,B 0,C 180,E1 -12334.304,E2 -12334.304} C_VEL
LIN {X 0,Y 374.592,Z 773.258,A -85,B 0,C 180,E1 -12336.077,E2 -12336.077} C_VEL
LIN {X 0,Y 374.766,Z 769.586,A -85,B 0,C 180,E1 -12337.543,E2 -12337.543} C_VEL
LIN {X 0,Y 375.13,Z 763.477,A -85,B 0,C 180,E1 -12339.435,E2 -12339.435} C_VEL
LIN {X 0,Y 375.655,Z 756.777,A -85,B 0,C 180,E1 -12341.055,E2 -12341.055} C_VEL
LIN {X 0,Y 376.513,Z 748.479,A -85,B 0,C 180,E1 -12342.669,E2 -12342.669} C_VEL
LIN {X 0,Y 377.348,Z 740.019,A -85,B 0,C 180,E1 -12344.011,E2 -12344.011} C_VEL
LIN {X 0,Y 378.236,Z 730.81,A -85,B 0,C 180,E1 -12345.216,E2 -12345.216} C_VEL
LIN {X 0,Y 379.273,Z 719.398,A -85,B 0,C 180,E1 -12346.414,E2 -12346.414} C_VEL
LIN {X 0,Y 380.298,Z 708.258,A -85,B 0,C 180,E1 -12347.337,E2 -12347.337} C_VEL
LIN {X 0,Y 381.25,Z 695.937,A -85,B 0,C 180,E1 -12348.124,E2 -12348.124} C_VEL
LIN {X 0,Y 382.046,Z 683.017,A -85,B 0,C 180,E1 -12348.709,E2 -12348.709} C_VEL
LIN {X 0,Y 382.644,Z 669.533,A -85,B 0,C 180,E1 -12349.096,E2 -12349.096} C_VEL
LIN {X 0,Y 383.761,Z 600.332,A -85,B 0,C 180,E1 -12350.48,E2 -12350.48} C_VEL
LIN {X 0,Y 380.384,Z 576.305,A -85,B 0,C 180,E1 -12351.201,E2 -12351.201} C_VEL
LIN {X 0,Y 378.461,Z 565.172,A -85,B 0,C 180,E1 -12351.576,E2 -12351.576} C_VEL
LIN {X 0,Y 380.346,Z 545.352,A -85,B 0,C 180,E1 -12355.736,E2 -12355.736} C_VEL
LIN {X 0,Y 380.105,Z 541.56,A -85,B 0,C 180,E1 -12356.587,E2 -12356.587} C_VEL
LIN {X 0,Y 377.978,Z 531.182,A -85,B 0,C 180,E1 -12359.084,E2 -12359.084} C_VEL
LIN {X 0,Y 375.96,Z 522.658,A -85,B 0,C 180,E1 -12361.268,E2 -12361.268} C_VEL
LIN {X 0,Y 375.98,Z 522.657,A -85,B 0,C 180,E1 -12364.666,E2 -12364.666} C_VEL
LIN {X 0,Y 375.977,Z 522.654,A -85,B 0,C 180,E1 -12368.27,E2 -12368.27} C_VEL
LIN {X 0,Y 375.988,Z 522.649,A -85,B 0,C 180,E1 -12371.609,E2 -12371.609} C_VEL
LIN {X 0,Y 375.968,Z 522.651,A -85,B 0,C 180,E1 -12375.261,E2 -12375.261} C_VEL
LIN {X 0,Y 375.938,Z 522.656,A -85,B 0,C 180,E1 -12379.132,E2 -12379.132} C_VEL
LIN {X 0,Y 375.962,Z 522.652,A -85,B 0,C 180,E1 -12381.911,E2 -12381.911} C_VEL
LIN {X 0,Y 375.976,Z 522.648,A -85,B 0,C 180,E1 -12385.332,E2 -12385.332} C_VEL
LIN {X 0,Y 375.955,Z 522.655,A -85,B 0,C 180,E1 -12388.437,E2 -12388.437} C_VEL
LIN {X 0,Y 375.997,Z 522.645,A -85,B 0,C 180,E1 -12392.141,E2 -12392.141} C_VEL
LIN {X 0,Y 376.001,Z 522.65,A -85,B 0,C 180,E1 -12394.538,E2 -12394.538} C_VEL
LIN {X 0,Y 375.957,Z 522.652,A -85,B 0,C 180,E1 -12398.045,E2 -12398.045} C_VEL
LIN {X 0,Y 376.002,Z 522.646,A -85,B 0,C 180,E1 -12401.472,E2 -12401.472} C_VEL
LIN {X 0,Y 376.052,Z 522.645,A -85,B 0,C 180,E1 -12404.832,E2 -12404.832} C_VEL
LIN {X 0,Y 376.043,Z 522.641,A -85,B 0,C 180,E1 -12408.136,E2 -12408.136} C_VEL
LIN {X 0,Y 376.212,Z 522.62,A -85,B 0,C 180,E1 -12411.917,E2 -12411.917} C_VEL
LIN {X 0,Y 376.17,Z 522.624,A -85,B 0,C 180,E1 -12414.639,E2 -12414.639} C_VEL
LIN {X 0,Y 376.346,Z 522.602,A -85,B 0,C 180,E1 -12417.859,E2 -12417.859} C_VEL
LIN {X 0,Y 376.482,Z 522.584,A -85,B 0,C 180,E1 -12419.999,E2 -12419.999} C_VEL
LIN {X 0,Y 376.184,Z 522.624,A -85,B 0,C 180,E1 -12423.212,E2 -12423.212} C_VEL
LIN {X 0,Y 376.228,Z 522.617,A -85,B 0,C 180,E1 -12426.572,E2 -12426.572} C_VEL
LIN {X 0,Y 376.111,Z 522.635,A -85,B 0,C 180,E1 -12429.681,E2 -12429.681} C_VEL
LIN {X 0,Y 376.08,Z 522.638,A -85,B 0,C 180,E1 -12433.657,E2 -12433.657} C_VEL
LIN {X 0,Y 376.034,Z 522.645,A -85,B 0,C 180,E1 -12437.607,E2 -12437.607} C_VEL
LIN {X 0,Y 375.969,Z 522.654,A -85,B 0,C 180,E1 -12440.832,E2 -12440.832} C_VEL
LIN {X 0,Y 375.985,Z 522.655,A -85,B 0,C 180,E1 -12444.281,E2 -12444.281} C_VEL
LIN {X 0,Y 376.011,Z 522.653,A -85,B 0,C 180,E1 -12446.652,E2 -12446.652} C_VEL
LIN {X 0,Y 376.021,Z 522.763,A -85,B 0,C 180,E1 -12448.713,E2 -12448.713} C_VEL
LIN {X 0,Y 377.177,Z 528.34,A -85,B 0,C 180,E1 -12450.431,E2 -12450.431} C_VEL
LIN {X 0,Y 383.663,Z 544.871,A -85,B 0,C 180,E1 -12451.22,E2 -12451.22} C_VEL
LIN {X 0,Y 384.64,Z 549.476,A -85,B 0,C 180,E1 -12451.381,E2 -12451.381} C_VEL
LIN {X 0,Y 382.914,Z 634.549,A -85,B 0,C 180,E1 -12453.099,E2 -12453.099} C_VEL
LIN {X 0,Y 382.395,Z 648.379,A -85,B 0,C 180,E1 -12453.609,E2 -12453.609} C_VEL
LIN {X 0,Y 381.856,Z 660.334,A -85,B 0,C 180,E1 -12454.264,E2 -12454.264} C_VEL
LIN {X 0,Y 380.968,Z 672.433,A -85,B 0,C 180,E1 -12455.15,E2 -12455.15} C_VEL
LIN {X 0,Y 379.989,Z 684.375,A -85,B 0,C 180,E1 -12456.288,E2 -12456.288} C_VEL
LIN {X 0,Y 378.948,Z 695.037,A -85,B 0,C 180,E1 -12457.579,E2 -12457.579} C_VEL
LIN {X 0,Y 378.01,Z 703.878,A -85,B 0,C 180,E1 -12458.904,E2 -12458.904} C_VEL
LIN {X 0,Y 377.047,Z 712.563,A -85,B 0,C 180,E1 -12460.511,E2 -12460.511} C_VEL
LIN {X 0,Y 376.231,Z 719.987,A -85,B 0,C 180,E1 -12462.258,E2 -12462.258} C_VEL
LIN {X 0,Y 375.578,Z 726.467,A -85,B 0,C 180,E1 -12464.234,E2 -12464.234} C_VEL
LIN {X 0,Y 375.133,Z 731.002,A -85,B 0,C 180,E1 -12466.119,E2 -12466.119} C_VEL
LIN {X 0,Y 374.856,Z 733.531,A -85,B 0,C 180,E1 -12467.551,E2 -12467.551} C_VEL
LIN {X 0,Y 374.649,Z 735.245,A -85,B 0,C 180,E1 -12468.963,E2 -12468.963} C_VEL
LIN {X 0,Y 374.494,Z 736.276,A -85,B 0,C 180,E1 -12470.353,E2 -12470.353} C_VEL
LIN {X 0,Y 374.462,Z 736.623,A -85,B 0,C 180,E1 -12472.023,E2 -12472.023} C_VEL
LIN {X 0,Y 374.499,Z 735.93,A -85,B 0,C 180,E1 -12473.798,E2 -12473.798} C_VEL
LIN {X 0,Y 374.679,Z 733.887,A -85,B 0,C 180,E1 -12475.757,E2 -12475.757} C_VEL
LIN {X 0,Y 374.961,Z 730.894,A -85,B 0,C 180,E1 -12477.505,E2 -12477.505} C_VEL
LIN {X 0,Y 375.375,Z 726.151,A -85,B 0,C 180,E1 -12479.455,E2 -12479.455} C_VEL
LIN {X 0,Y 375.904,Z 720.305,A -85,B 0,C 180,E1 -12481.232,E2 -12481.232} C_VEL
LIN {X 0,Y 376.458,Z 713.883,A -85,B 0,C 180,E1 -12482.782,E2 -12482.782} C_VEL
LIN {X 0,Y 377.206,Z 705.951,A -85,B 0,C 180,E1 -12484.331,E2 -12484.331} C_VEL
LIN {X 0,Y 378.004,Z 697.688,A -85,B 0,C 180,E1 -12485.646,E2 -12485.646} C_VEL
LIN {X 0,Y 378.878,Z 687.793,A -85,B 0,C 180,E1 -12486.93,E2 -12486.93} C_VEL
LIN {X 0,Y 379.793,Z 676.343,A -85,B 0,C 180,E1 -12488.116,E2 -12488.116} C_VEL
LIN {X 0,Y 380.619,Z 664.079,A -85,B 0,C 180,E1 -12489.109,E2 -12489.109} C_VEL
LIN {X 0,Y 381.266,Z 652.597,A -85,B 0,C 180,E1 -12489.81,E2 -12489.81} C_VEL
LIN {X 0,Y 381.743,Z 640.137,A -85,B 0,C 180,E1 -12490.362,E2 -12490.362} C_VEL
LIN {X 0,Y 382.063,Z 627.122,A -85,B 0,C 180,E1 -12490.729,E2 -12490.729} C_VEL
LIN {X 0,Y 383.323,Z 547.522,A -85,B 0,C 180,E1 -12492.293,E2 -12492.293} C_VEL
LIN {X 0,Y 380.972,Z 538.609,A -85,B 0,C 180,E1 -12492.6,E2 -12492.6} C_VEL
LIN {X 0,Y 376.781,Z 526.412,A -85,B 0,C 180,E1 -12493.091,E2 -12493.091} C_VEL
LIN {X 0,Y 376.05,Z 522.642,A -85,B 0,C 180,E1 -12494.208,E2 -12494.208} C_VEL
LIN {X 0,Y 376.107,Z 522.636,A -85,B 0,C 180,E1 -12497.042,E2 -12497.042} C_VEL
LIN {X 0,Y 376.116,Z 522.632,A -85,B 0,C 180,E1 -12500.319,E2 -12500.319} C_VEL
LIN {X 0,Y 376.235,Z 522.616,A -85,B 0,C 180,E1 -12503.565,E2 -12503.565} C_VEL
LIN {X 0,Y 376.351,Z 522.601,A -85,B 0,C 180,E1 -12507.86,E2 -12507.86} C_VEL
LIN {X 0,Y 376.486,Z 522.584,A -85,B 0,C 180,E1 -12510,E2 -12510} C_VEL
LIN {X 0,Y 376.281,Z 522.615,A -85,B 0,C 180,E1 -12511.076,E2 -12511.076} C_VEL
LIN {X 0,Y 375.609,Z 522.694,A -85,B 0,C 180,E1 -12511.967,E2 -12511.967} C_VEL
LIN {X 0,Y 372.704,Z 523.057,A -85,B 0,C 180,E1 -12513.416,E2 -12513.416} C_VEL
LIN {X 0,Y 370.254,Z 523.364,A -85,B 0,C 180,E1 -12514.587,E2 -12514.587} C_VEL
LIN {X 0,Y 369.221,Z 523.491,A -85,B 0,C 180,E1 -12515.494,E2 -12515.494} C_VEL
LIN {X 0,Y 369.147,Z 523.499,A -85,B 0,C 180,E1 -12515.801,E2 -12515.801} C_VEL
LIN {X 0,Y 369.135,Z 523.505,A -85,B 0,C 180,E1 -12518.761,E2 -12518.761} C_VEL
LIN {X 0,Y 369.002,Z 523.517,A -85,B 0,C 180,E1 -12522.093,E2 -12522.093} C_VEL
LIN {X 0,Y 368.994,Z 523.519,A -85,B 0,C 180,E1 -12525.465,E2 -12525.465} C_VEL
LIN {X 0,Y 368.954,Z 523.528,A -85,B 0,C 180,E1 -12528.894,E2 -12528.894} C_VEL
LIN {X 0,Y 368.928,Z 523.527,A -85,B 0,C 180,E1 -12532.395,E2 -12532.395} C_VEL
LIN {X 0,Y 368.995,Z 523.517,A -85,B 0,C 180,E1 -12535.98,E2 -12535.98} C_VEL
LIN {X 0,Y 368.963,Z 523.526,A -85,B 0,C 180,E1 -12538.813,E2 -12538.813} C_VEL
LIN {X 0,Y 368.905,Z 523.529,A -85,B 0,C 180,E1 -12542.236,E2 -12542.236} C_VEL
LIN {X 0,Y 368.924,Z 523.533,A -85,B 0,C 180,E1 -12545.001,E2 -12545.001} C_VEL
LIN {X 0,Y 368.908,Z 523.531,A -85,B 0,C 180,E1 -12548.641,E2 -12548.641} C_VEL
LIN {X 0,Y 368.935,Z 523.525,A -85,B 0,C 180,E1 -12552.02,E2 -12552.02} C_VEL
LIN {X 0,Y 368.982,Z 523.524,A -85,B 0,C 180,E1 -12555.192,E2 -12555.192} C_VEL
LIN {X 0,Y 368.934,Z 523.525,A -85,B 0,C 180,E1 -12558.185,E2 -12558.185} C_VEL
LIN {X 0,Y 368.906,Z 523.532,A -85,B 0,C 180,E1 -12561.358,E2 -12561.358} C_VEL
LIN {X 0,Y 368.929,Z 523.532,A -85,B 0,C 180,E1 -12565.146,E2 -12565.146} C_VEL
LIN {X 0,Y 368.921,Z 523.533,A -85,B 0,C 180,E1 -12569.046,E2 -12569.046} C_VEL
LIN {X 0,Y 368.978,Z 523.522,A -85,B 0,C 180,E1 -12571.564,E2 -12571.564} C_VEL
LIN {X 0,Y 368.991,Z 523.518,A -85,B 0,C 180,E1 -12574.02,E2 -12574.02} C_VEL
LIN {X 0,Y 368.916,Z 523.529,A -85,B 0,C 180,E1 -12577.604,E2 -12577.604} C_VEL
LIN {X 0,Y 368.949,Z 523.53,A -85,B 0,C 180,E1 -12581.106,E2 -12581.106} C_VEL
LIN {X 0,Y 368.989,Z 523.519,A -85,B 0,C 180,E1 -12584.535,E2 -12584.535} C_VEL
LIN {X 0,Y 369.004,Z 523.517,A -85,B 0,C 180,E1 -12587.907,E2 -12587.907} C_VEL
LIN {X 0,Y 369.221,Z 523.49,A -85,B 0,C 180,E1 -12591.801,E2 -12591.801} C_VEL
LIN {X 0,Y 369.143,Z 523.5,A -85,B 0,C 180,E1 -12594.538,E2 -12594.538} C_VEL
LIN {X 0,Y 369.311,Z 523.479,A -85,B 0,C 180,E1 -12597.819,E2 -12597.819} C_VEL
LIN {X 0,Y 369.452,Z 523.461,A -85,B 0,C 180,E1 -12600.001,E2 -12600.001} C_VEL
LIN {X 0,Y 369.317,Z 523.477,A -85,B 0,C 180,E1 -12602.182,E2 -12602.182} C_VEL
LIN {X 0,Y 369.2,Z 523.493,A -85,B 0,C 180,E1 -12606.559,E2 -12606.559} C_VEL
LIN {X 0,Y 369.06,Z 523.51,A -85,B 0,C 180,E1 -12609.869,E2 -12609.869} C_VEL
LIN {X 0,Y 369.03,Z 523.515,A -85,B 0,C 180,E1 -12613.773,E2 -12613.773} C_VEL
LIN {X 0,Y 368.995,Z 523.519,A -85,B 0,C 180,E1 -12617.769,E2 -12617.769} C_VEL
LIN {X 0,Y 368.923,Z 523.533,A -85,B 0,C 180,E1 -12621.221,E2 -12621.221} C_VEL
LIN {X 0,Y 368.952,Z 523.525,A -85,B 0,C 180,E1 -12624.776,E2 -12624.776} C_VEL
LIN {X 0,Y 368.982,Z 523.519,A -85,B 0,C 180,E1 -12628.436,E2 -12628.436} C_VEL
LIN {X 0,Y 368.905,Z 523.529,A -85,B 0,C 180,E1 -12632.238,E2 -12632.238} C_VEL
LIN {X 0,Y 368.925,Z 523.529,A -85,B 0,C 180,E1 -12635.002,E2 -12635.002} C_VEL
LIN {X 0,Y 368.907,Z 523.529,A -85,B 0,C 180,E1 -12638.642,E2 -12638.642} C_VEL
LIN {X 0,Y 368.879,Z 523.533,A -85,B 0,C 180,E1 -12642.011,E2 -12642.011} C_VEL
LIN {X 0,Y 368.952,Z 523.528,A -85,B 0,C 180,E1 -12645.188,E2 -12645.188} C_VEL
LIN {X 0,Y 368.939,Z 523.525,A -85,B 0,C 180,E1 -12648.187,E2 -12648.187} C_VEL
LIN {X 0,Y 368.913,Z 523.535,A -85,B 0,C 180,E1 -12651.36,E2 -12651.36} C_VEL
LIN {X 0,Y 368.937,Z 523.529,A -85,B 0,C 180,E1 -12655.147,E2 -12655.147} C_VEL
LIN {X 0,Y 368.937,Z 523.59,A -85,B 0,C 180,E1 -12659.048,E2 -12659.048} C_VEL
LIN {X 0,Y 372.135,Z 538.301,A -85,B 0,C 180,E1 -12662.577,E2 -12662.577} C_VEL
LIN {X 0,Y 373.156,Z 544.647,A -85,B 0,C 180,E1 -12664.031,E2 -12664.031} C_VEL
LIN {X 0,Y 371.683,Z 561.019,A -85,B 0,C 180,E1 -12667.487,E2 -12667.487} C_VEL
LIN {X 0,Y 371.26,Z 566.437,A -85,B 0,C 180,E1 -12668.62,E2 -12668.62} C_VEL
LIN {X 0,Y 376.097,Z 601.427,A -85,B 0,C 180,E1 -12669.615,E2 -12669.615} C_VEL
LIN {X 0,Y 374.863,Z 675.759,A -85,B 0,C 180,E1 -12671.131,E2 -12671.131} C_VEL
LIN {X 0,Y 374.125,Z 689.404,A -85,B 0,C 180,E1 -12671.625,E2 -12671.625} C_VEL
LIN {X 0,Y 373.252,Z 702.3,A -85,B 0,C 180,E1 -12672.325,E2 -12672.325} C_VEL
LIN {X 0,Y 372.312,Z 714.891,A -85,B 0,C 180,E1 -12673.27,E2 -12673.27} C_VEL
LIN {X 0,Y 371.259,Z 726.135,A -85,B 0,C 180,E1 -12674.351,E2 -12674.351} C_VEL
LIN {X 0,Y 370.313,Z 737.257,A -85,B 0,C 180,E1 -12675.717,E2 -12675.717} C_VEL
LIN {X 0,Y 369.451,Z 746.258,A -85,B 0,C 180,E1 -12677.085,E2 -12677.085} C_VEL
LIN {X 0,Y 368.594,Z 755.037,A -85,B 0,C 180,E1 -12678.73,E2 -12678.73} C_VEL
LIN {X 0,Y 368.081,Z 762.04,A -85,B 0,C 180,E1 -12680.383,E2 -12680.383} C_VEL
LIN {X 0,Y 367.694,Z 768.461,A -85,B 0,C 180,E1 -12682.311,E2 -12682.311} C_VEL
LIN {X 0,Y 367.545,Z 772.491,A -85,B 0,C 180,E1 -12683.892,E2 -12683.892} C_VEL
LIN {X 0,Y 367.515,Z 775.761,A -85,B 0,C 180,E1 -12685.613,E2 -12685.613} C_VEL
LIN {X 0,Y 367.474,Z 777.291,A -85,B 0,C 180,E1 -12686.711,E2 -12686.711} C_VEL
LIN {X 0,Y 367.588,Z 778.363,A -85,B 0,C 180,E1 -12687.809,E2 -12687.809} C_VEL
LIN {X 0,Y 367.597,Z 779.021,A -85,B 0,C 180,E1 -12688.905,E2 -12688.905} C_VEL
LIN {X 0,Y 367.578,Z 779.279,A -85,B 0,C 180,E1 -12690,E2 -12690} C_VEL
LIN {X 0,Y 367.596,Z 779.136,A -85,B 0,C 180,E1 -12691.095,E2 -12691.095} C_VEL
LIN {X 0,Y 367.567,Z 778.545,A -85,B 0,C 180,E1 -12692.192,E2 -12692.192} C_VEL
LIN {X 0,Y 367.504,Z 776.151,A -85,B 0,C 180,E1 -12694.387,E2 -12694.387} C_VEL
LIN {X 0,Y 367.49,Z 773.234,A -85,B 0,C 180,E1 -12696.027,E2 -12696.027} C_VEL
LIN {X 0,Y 367.693,Z 769.237,A -85,B 0,C 180,E1 -12697.689,E2 -12697.689} C_VEL
LIN {X 0,Y 368.001,Z 764.115,A -85,B 0,C 180,E1 -12699.342,E2 -12699.342} C_VEL
LIN {X 0,Y 368.507,Z 757.703,A -85,B 0,C 180,E1 -12700.994,E2 -12700.994} C_VEL
LIN {X 0,Y 369.382,Z 749.705,A -85,B 0,C 180,E1 -12702.638,E2 -12702.638} C_VEL
LIN {X 0,Y 370.223,Z 741.564,A -85,B 0,C 180,E1 -12704.006,E2 -12704.006} C_VEL
LIN {X 0,Y 371.249,Z 731.678,A -85,B 0,C 180,E1 -12705.368,E2 -12705.368} C_VEL
LIN {X 0,Y 372.328,Z 720.703,A -85,B 0,C 180,E1 -12706.588,E2 -12706.588} C_VEL
LIN {X 0,Y 373.532,Z 708.23,A -85,B 0,C 180,E1 -12707.661,E2 -12707.661} C_VEL
LIN {X 0,Y 374.533,Z 696.059,A -85,B 0,C 180,E1 -12708.46,E2 -12708.46} C_VEL
LIN {X 0,Y 375.347,Z 683.472,A -85,B 0,C 180,E1 -12709.056,E2 -12709.056} C_VEL
LIN {X 0,Y 375.989,Z 670.544,A -85,B 0,C 180,E1 -12709.448,E2 -12709.448} C_VEL
LIN {X 0,Y 377.135,Z 600.908,A -85,B 0,C 180,E1 -12710.875,E2 -12710.875} C_VEL
LIN {X 0,Y 373.777,Z 577.005,A -85,B 0,C 180,E1 -12711.613,E2 -12711.613} C_VEL
LIN {X 0,Y 371.652,Z 564.74,A -85,B 0,C 180,E1 -12712.033,E2 -12712.033} C_VEL
LIN {X 0,Y 373.492,Z 546.51,A -85,B 0,C 180,E1 -12715.943,E2 -12715.943} C_VEL
LIN {X 0,Y 373.09,Z 542.487,A -85,B 0,C 180,E1 -12716.877,E2 -12716.877} C_VEL
LIN {X 0,Y 370.886,Z 531.827,A -85,B 0,C 180,E1 -12719.516,E2 -12719.516} C_VEL
LIN {X 0,Y 368.921,Z 523.535,A -85,B 0,C 180,E1 -12721.712,E2 -12721.712} C_VEL
LIN {X 0,Y 368.929,Z 523.536,A -85,B 0,C 180,E1 -12725.001,E2 -12725.001} C_VEL
LIN {X 0,Y 368.912,Z 523.533,A -85,B 0,C 180,E1 -12728.64,E2 -12728.64} C_VEL
LIN {X 0,Y 368.94,Z 523.528,A -85,B 0,C 180,E1 -12732.019,E2 -12732.019} C_VEL
LIN {X 0,Y 368.922,Z 523.528,A -85,B 0,C 180,E1 -12735.182,E2 -12735.182} C_VEL
LIN {X 0,Y 368.88,Z 523.531,A -85,B 0,C 180,E1 -12738.177,E2 -12738.177} C_VEL
LIN {X 0,Y 368.907,Z 523.532,A -85,B 0,C 180,E1 -12741.358,E2 -12741.358} C_VEL
LIN {X 0,Y 368.933,Z 523.526,A -85,B 0,C 180,E1 -12745.145,E2 -12745.145} C_VEL
LIN {X 0,Y 368.925,Z 523.527,A -85,B 0,C 180,E1 -12749.045,E2 -12749.045} C_VEL
LIN {X 0,Y 368.982,Z 523.519,A -85,B 0,C 180,E1 -12751.564,E2 -12751.564} C_VEL
LIN {X 0,Y 368.952,Z 523.521,A -85,B 0,C 180,E1 -12755.224,E2 -12755.224} C_VEL
LIN {X 0,Y 368.931,Z 523.525,A -85,B 0,C 180,E1 -12758.972,E2 -12758.972} C_VEL
LIN {X 0,Y 368.984,Z 523.52,A -85,B 0,C 180,E1 -12762.256,E2 -12762.256} C_VEL
LIN {X 0,Y 369.03,Z 523.513,A -85,B 0,C 180,E1 -12766.227,E2 -12766.227} C_VEL
LIN {X 0,Y 369.06,Z 523.507,A -85,B 0,C 180,E1 -12770.131,E2 -12770.131} C_VEL
LIN {X 0,Y 369.156,Z 523.5,A -85,B 0,C 180,E1 -12772.341,E2 -12772.341} C_VEL
LIN {X 0,Y 369.142,Z 523.498,A -85,B 0,C 180,E1 -12774.537,E2 -12774.537} C_VEL
LIN {X 0,Y 369.311,Z 523.479,A -85,B 0,C 180,E1 -12777.818,E2 -12777.818} C_VEL
LIN {X 0,Y 369.452,Z 523.46,A -85,B 0,C 180,E1 -12779.999,E2 -12779.999} C_VEL
LIN {X 0,Y 369.311,Z 523.481,A -85,B 0,C 180,E1 -12782.181,E2 -12782.181} C_VEL
LIN {X 0,Y 369.199,Z 523.493,A -85,B 0,C 180,E1 -12786.558,E2 -12786.558} C_VEL
LIN {X 0,Y 369.059,Z 523.512,A -85,B 0,C 180,E1 -12789.868,E2 -12789.868} C_VEL
LIN {X 0,Y 369.028,Z 523.516,A -85,B 0,C 180,E1 -12793.772,E2 -12793.772} C_VEL
LIN {X 0,Y 368.993,Z 523.522,A -85,B 0,C 180,E1 -12797.768,E2 -12797.768} C_VEL
LIN {X 0,Y 368.92,Z 523.534,A -85,B 0,C 180,E1 -12801.22,E2 -12801.22} C_VEL
LIN {X 0,Y 368.949,Z 523.531,A -85,B 0,C 180,E1 -12804.775,E2 -12804.775} C_VEL
LIN {X 0,Y 368.945,Z 523.553,A -85,B 0,C 180,E1 -12808.283,E2 -12808.283} C_VEL
LIN {X 0,Y 370.084,Z 528.843,A -85,B 0,C 180,E1 -12809.939,E2 -12809.939} C_VEL
LIN {X 0,Y 377.105,Z 546.346,A -85,B 0,C 180,E1 -12810.823,E2 -12810.823} C_VEL
LIN {X 0,Y 378.1,Z 550.276,A -85,B 0,C 180,E1 -12810.976,E2 -12810.976} C_VEL
LIN {X 0,Y 376.301,Z 635.255,A -85,B 0,C 180,E1 -12812.729,E2 -12812.729} C_VEL
LIN {X 0,Y 375.764,Z 648.905,A -85,B 0,C 180,E1 -12813.243,E2 -12813.243} C_VEL
LIN {X 0,Y 375.169,Z 661.099,A -85,B 0,C 180,E1 -12813.925,E2 -12813.925} C_VEL
LIN {X 0,Y 374.265,Z 672.854,A -85,B 0,C 180,E1 -12814.804,E2 -12814.804} C_VEL
LIN {X 0,Y 373.257,Z 684.609,A -85,B 0,C 180,E1 -12815.941,E2 -12815.941} C_VEL
LIN {X 0,Y 372.247,Z 694.686,A -85,B 0,C 180,E1 -12817.168,E2 -12817.168} C_VEL
LIN {X 0,Y 371.125,Z 704.59,A -85,B 0,C 180,E1 -12818.676,E2 -12818.676} C_VEL
LIN {X 0,Y 370.18,Z 712.681,A -85,B 0,C 180,E1 -12820.202,E2 -12820.202} C_VEL
LIN {X 0,Y 369.372,Z 719.34,A -85,B 0,C 180,E1 -12821.754,E2 -12821.754} C_VEL
LIN {X 0,Y 368.686,Z 725.525,A -85,B 0,C 180,E1 -12823.585,E2 -12823.585} C_VEL
LIN {X 0,Y 368.306,Z 729.505,A -85,B 0,C 180,E1 -12825.088,E2 -12825.088} C_VEL
LIN {X 0,Y 367.967,Z 732.535,A -85,B 0,C 180,E1 -12826.562,E2 -12826.562} C_VEL
LIN {X 0,Y 367.676,Z 734.946,A -85,B 0,C 180,E1 -12828.199,E2 -12828.199} C_VEL
LIN {X 0,Y 367.47,Z 736.48,A -85,B 0,C 180,E1 -12829.907,E2 -12829.907} C_VEL
LIN {X 0,Y 367.37,Z 737.04,A -85,B 0,C 180,E1 -12831.66,E2 -12831.66} C_VEL
LIN {X 0,Y 367.433,Z 736.461,A -85,B 0,C 180,E1 -12833.635,E2 -12833.635} C_VEL
LIN {X 0,Y 367.551,Z 734.944,A -85,B 0,C 180,E1 -12835.305,E2 -12835.305} C_VEL
LIN {X 0,Y 367.814,Z 732.01,A -85,B 0,C 180,E1 -12837.216,E2 -12837.216} C_VEL
LIN {X 0,Y 368.245,Z 727.56,A -85,B 0,C 180,E1 -12839.184,E2 -12839.184} C_VEL
LIN {X 0,Y 368.68,Z 722.724,A -85,B 0,C 180,E1 -12840.797,E2 -12840.797} C_VEL
LIN {X 0,Y 369.323,Z 716.195,A -85,B 0,C 180,E1 -12842.519,E2 -12842.519} C_VEL
LIN {X 0,Y 370.021,Z 708.702,A -85,B 0,C 180,E1 -12844.098,E2 -12844.098} C_VEL
LIN {X 0,Y 370.988,Z 699.069,A -85,B 0,C 180,E1 -12845.717,E2 -12845.717} C_VEL
LIN {X 0,Y 371.859,Z 689.365,A -85,B 0,C 180,E1 -12847.036,E2 -12847.036} C_VEL
LIN {X 0,Y 372.741,Z 679.307,A -85,B 0,C 180,E1 -12848.138,E2 -12848.138} C_VEL
LIN {X 0,Y 373.596,Z 667.429,A -85,B 0,C 180,E1 -12849.17,E2 -12849.17} C_VEL
LIN {X 0,Y 374.342,Z 655.084,A -85,B 0,C 180,E1 -12849.993,E2 -12849.993} C_VEL
LIN {X 0,Y 374.89,Z 642.348,A -85,B 0,C 180,E1 -12850.6,E2 -12850.6} C_VEL
LIN {X 0,Y 375.243,Z 628.916,A -85,B 0,C 180,E1 -12851.009,E2 -12851.009} C_VEL
LIN {X 0,Y 376.735,Z 549.151,A -85,B 0,C 180,E1 -12852.603,E2 -12852.603} C_VEL
LIN {X 0,Y 374.32,Z 540.146,A -85,B 0,C 180,E1 -12852.923,E2 -12852.923} C_VEL
LIN {X 0,Y 369.621,Z 526.738,A -85,B 0,C 180,E1 -12853.5,E2 -12853.5} C_VEL
LIN {X 0,Y 369.013,Z 523.52,A -85,B 0,C 180,E1 -12854.465,E2 -12854.465} C_VEL
LIN {X 0,Y 369.064,Z 523.515,A -85,B 0,C 180,E1 -12856.791,E2 -12856.791} C_VEL
LIN {X 0,Y 369.064,Z 523.509,A -85,B 0,C 180,E1 -12860.132,E2 -12860.132} C_VEL
LIN {X 0,Y 369.158,Z 523.499,A -85,B 0,C 180,E1 -12862.342,E2 -12862.342} C_VEL
LIN {X 0,Y 369.139,Z 523.502,A -85,B 0,C 180,E1 -12864.538,E2 -12864.538} C_VEL
LIN {X 0,Y 369.316,Z 523.478,A -85,B 0,C 180,E1 -12867.819,E2 -12867.819} C_VEL
LIN {X 0,Y 369.456,Z 523.46,A -85,B 0,C 180,E1 -12870,E2 -12870} C_VEL
LIN {X 0,Y 369.316,Z 523.478,A -85,B 0,C 180,E1 -12872.181,E2 -12872.181} C_VEL
LIN {X 0,Y 369.147,Z 523.499,A -85,B 0,C 180,E1 -12875.801,E2 -12875.801} C_VEL
LIN {X 0,Y 368.503,Z 523.584,A -85,B 0,C 180,E1 -12876.712,E2 -12876.712} C_VEL
LIN {X 0,Y 365.627,Z 523.938,A -85,B 0,C 180,E1 -12878.193,E2 -12878.193} C_VEL
LIN {X 0,Y 363.159,Z 524.247,A -85,B 0,C 180,E1 -12879.39,E2 -12879.39} C_VEL
LIN {X 0,Y 362.078,Z 524.38,A -85,B 0,C 180,E1 -12880.317,E2 -12880.317} C_VEL
LIN {X 0,Y 361.981,Z 524.391,A -85,B 0,C 180,E1 -12880.632,E2 -12880.632} C_VEL
LIN {X 0,Y 361.994,Z 524.39,A -85,B 0,C 180,E1 -12883.899,E2 -12883.899} C_VEL
LIN {X 0,Y 361.963,Z 524.393,A -85,B 0,C 180,E1 -12887.938,E2 -12887.938} C_VEL
LIN {X 0,Y 361.888,Z 524.404,A -85,B 0,C 180,E1 -12891.653,E2 -12891.653} C_VEL
LIN {X 0,Y 361.924,Z 524.402,A -85,B 0,C 180,E1 -12895.29,E2 -12895.29} C_VEL
LIN {X 0,Y 361.918,Z 524.399,A -85,B 0,C 180,E1 -12897.777,E2 -12897.777} C_VEL
LIN {X 0,Y 361.855,Z 524.408,A -85,B 0,C 180,E1 -12901.627,E2 -12901.627} C_VEL
LIN {X 0,Y 361.869,Z 524.409,A -85,B 0,C 180,E1 -12905.345,E2 -12905.345} C_VEL
LIN {X 0,Y 361.87,Z 524.412,A -85,B 0,C 180,E1 -12909.028,E2 -12909.028} C_VEL
LIN {X 0,Y 361.88,Z 524.405,A -85,B 0,C 180,E1 -12912.44,E2 -12912.44} C_VEL
LIN {X 0,Y 361.921,Z 524.399,A -85,B 0,C 180,E1 -12915.928,E2 -12915.928} C_VEL
LIN {X 0,Y 361.898,Z 524.406,A -85,B 0,C 180,E1 -12919.232,E2 -12919.232} C_VEL
LIN {X 0,Y 361.862,Z 524.412,A -85,B 0,C 180,E1 -12922.982,E2 -12922.982} C_VEL
LIN {X 0,Y 361.851,Z 524.409,A -85,B 0,C 180,E1 -12926.631,E2 -12926.631} C_VEL
LIN {X 0,Y 361.868,Z 524.407,A -85,B 0,C 180,E1 -12929.672,E2 -12929.672} C_VEL
LIN {X 0,Y 361.946,Z 524.398,A -85,B 0,C 180,E1 -12933.475,E2 -12933.475} C_VEL
LIN {X 0,Y 361.873,Z 524.411,A -85,B 0,C 180,E1 -12937.144,E2 -12937.144} C_VEL
LIN {X 0,Y 361.898,Z 524.404,A -85,B 0,C 180,E1 -12940.723,E2 -12940.723} C_VEL
LIN {X 0,Y 361.924,Z 524.404,A -85,B 0,C 180,E1 -12943.066,E2 -12943.066} C_VEL
LIN {X 0,Y 361.991,Z 524.391,A -85,B 0,C 180,E1 -12946.528,E2 -12946.528} C_VEL
LIN {X 0,Y 362.028,Z 524.386,A -85,B 0,C 180,E1 -12949.938,E2 -12949.938} C_VEL
LIN {X 0,Y 362.143,Z 524.371,A -85,B 0,C 180,E1 -12952.193,E2 -12952.193} C_VEL
LIN {X 0,Y 362.116,Z 524.375,A -85,B 0,C 180,E1 -12954.432,E2 -12954.432} C_VEL
LIN {X 0,Y 362.275,Z 524.356,A -85,B 0,C 180,E1 -12957.777,E2 -12957.777} C_VEL
LIN {X 0,Y 362.421,Z 524.337,A -85,B 0,C 180,E1 -12960.001,E2 -12960.001} C_VEL
LIN {X 0,Y 362.282,Z 524.354,A -85,B 0,C 180,E1 -12962.224,E2 -12962.224} C_VEL
LIN {X 0,Y 362.161,Z 524.37,A -85,B 0,C 180,E1 -12966.687,E2 -12966.687} C_VEL
LIN {X 0,Y 362.024,Z 524.386,A -85,B 0,C 180,E1 -12970.063,E2 -12970.063} C_VEL
LIN {X 0,Y 361.991,Z 524.391,A -85,B 0,C 180,E1 -12973.899,E2 -12973.899} C_VEL
LIN {X 0,Y 361.961,Z 524.394,A -85,B 0,C 180,E1 -12977.939,E2 -12977.939} C_VEL
LIN {X 0,Y 361.886,Z 524.406,A -85,B 0,C 180,E1 -12981.654,E2 -12981.654} C_VEL
LIN {X 0,Y 361.923,Z 524.405,A -85,B 0,C 180,E1 -12985.291,E2 -12985.291} C_VEL
LIN {X 0,Y 361.917,Z 524.401,A -85,B 0,C 180,E1 -12987.779,E2 -12987.779} C_VEL
LIN {X 0,Y 361.855,Z 524.41,A -85,B 0,C 180,E1 -12991.628,E2 -12991.628} C_VEL
LIN {X 0,Y 361.871,Z 524.412,A -85,B 0,C 180,E1 -12995.346,E2 -12995.346} C_VEL
LIN {X 0,Y 361.868,Z 524.409,A -85,B 0,C 180,E1 -12999.028,E2 -12999.028} C_VEL
LIN {X 0,Y 361.836,Z 524.411,A -85,B 0,C 180,E1 -13002.829,E2 -13002.829} C_VEL
LIN {X 0,Y 361.897,Z 524.403,A -85,B 0,C 180,E1 -13005.934,E2 -13005.934} C_VEL
LIN {X 0,Y 361.904,Z 524.406,A -85,B 0,C 180,E1 -13009.233,E2 -13009.233} C_VEL
LIN {X 0,Y 361.869,Z 524.408,A -85,B 0,C 180,E1 -13012.983,E2 -13012.983} C_VEL
LIN {X 0,Y 361.859,Z 524.411,A -85,B 0,C 180,E1 -13016.632,E2 -13016.632} C_VEL
LIN {X 0,Y 361.863,Z 524.414,A -85,B 0,C 180,E1 -13018.712,E2 -13018.712} C_VEL
LIN {X 0,Y 364.64,Z 537.054,A -85,B 0,C 180,E1 -13021.824,E2 -13021.824} C_VEL
LIN {X 0,Y 366.183,Z 545.453,A -85,B 0,C 180,E1 -13023.806,E2 -13023.806} C_VEL
LIN {X 0,Y 364.932,Z 559.092,A -85,B 0,C 180,E1 -13026.747,E2 -13026.747} C_VEL
LIN {X 0,Y 364.332,Z 566.03,A -85,B 0,C 180,E1 -13028.23,E2 -13028.23} C_VEL
LIN {X 0,Y 369.368,Z 602.345,A -85,B 0,C 180,E1 -13029.292,E2 -13029.292} C_VEL
LIN {X 0,Y 368.099,Z 675.252,A -85,B 0,C 180,E1 -13030.807,E2 -13030.807} C_VEL
LIN {X 0,Y 367.327,Z 688.922,A -85,B 0,C 180,E1 -13031.309,E2 -13031.309} C_VEL
LIN {X 0,Y 366.449,Z 701.326,A -85,B 0,C 180,E1 -13031.986,E2 -13031.986} C_VEL
LIN {X 0,Y 365.623,Z 712.461,A -85,B 0,C 180,E1 -13032.811,E2 -13032.811} C_VEL
LIN {X 0,Y 364.486,Z 724.07,A -85,B 0,C 180,E1 -13033.909,E2 -13033.909} C_VEL
LIN {X 0,Y 363.577,Z 734.342,A -85,B 0,C 180,E1 -13035.131,E2 -13035.131} C_VEL
LIN {X 0,Y 362.618,Z 743.98,A -85,B 0,C 180,E1 -13036.552,E2 -13036.552} C_VEL
LIN {X 0,Y 361.751,Z 753.098,A -85,B 0,C 180,E1 -13038.23,E2 -13038.23} C_VEL
LIN {X 0,Y 361.134,Z 760.443,A -85,B 0,C 180,E1 -13039.913,E2 -13039.913} C_VEL
LIN {X 0,Y 360.71,Z 766.305,A -85,B 0,C 180,E1 -13041.598,E2 -13041.598} C_VEL
LIN {X 0,Y 360.513,Z 770.907,A -85,B 0,C 180,E1 -13043.283,E2 -13043.283} C_VEL
LIN {X 0,Y 360.433,Z 773.322,A -85,B 0,C 180,E1 -13044.405,E2 -13044.405} C_VEL
LIN {X 0,Y 360.443,Z 775.298,A -85,B 0,C 180,E1 -13045.527,E2 -13045.527} C_VEL
LIN {X 0,Y 360.389,Z 776.842,A -85,B 0,C 180,E1 -13046.646,E2 -13046.646} C_VEL
